LIN {X 0,Y 411.383,Z 368.831,A -85,B 0,C 180,E1 -10541.579,E2 -10541.579} C_VEL
LIN {X 0,Y 411.988,Z 360.367,A -85,B 0,C 180,E1 -10542.812,E2 -10542.812} C_VEL
LIN {X 0,Y 412.688,Z 350.209,A -85,B 0,C 180,E1 -10544.018,E2 -10544.018} C_VEL
LIN {X 0,Y 413.617,Z 338.309,A -85,B 0,C 180,E1 -10545.143,E2 -10545.143} C_VEL
LIN {X 0,Y 414.492,Z 326.832,A -85,B 0,C 180,E1 -10545.993,E2 -10545.993} C_VEL
LIN {X 0,Y 414.334,Z 319.686,A -85,B 0,C 180,E1 -10546.442,E2 -10546.442} C_VEL
LIN {X 0,Y 412.96,Z 306.533,A -85,B 0,C 180,E1 -10547.145,E2 -10547.145} C_VEL
LIN {X 0,Y 410.807,Z 293.982,A -85,B 0,C 180,E1 -10547.664,E2 -10547.664} C_VEL
LIN {X 0,Y 410.419,Z 291.596,A -85,B 0,C 180,E1 -10547.758,E2 -10547.758} C_VEL
LIN {X 0,Y 410.785,Z 283.542,A -85,B 0,C 180,E1 -10551.055,E2 -10551.055} C_VEL
LIN {X 0,Y 411.122,Z 276.006,A -85,B 0,C 180,E1 -10554.221,E2 -10554.221} C_VEL
LIN {X 0,Y 411.591,Z 268.703,A -85,B 0,C 180,E1 -10557.386,E2 -10557.386} C_VEL
LIN {X 0,Y 412.207,Z 261.207,A -85,B 0,C 180,E1 -10560.762,E2 -10560.762} C_VEL
LIN {X 0,Y 412.806,Z 255.521,A -85,B 0,C 180,E1 -10563.463,E2 -10563.463} C_VEL
LIN {X 0,Y 413.225,Z 250.596,A -85,B 0,C 180,E1 -10565.926,E2 -10565.926} C_VEL
LIN {X 0,Y 412.966,Z 247.13,A -85,B 0,C 180,E1 -10567.781,E2 -10567.781} C_VEL
LIN {X 0,Y 412.21,Z 242.601,A -85,B 0,C 180,E1 -10570.381,E2 -10570.381} C_VEL
LIN {X 0,Y 411.179,Z 237.269,A -85,B 0,C 180,E1 -10573.842,E2 -10573.842} C_VEL
LIN {X 0,Y 411.181,Z 237.269,A -85,B 0,C 180,E1 -10577.303,E2 -10577.303} C_VEL
LIN {X 0,Y 411.218,Z 237.265,A -85,B 0,C 180,E1 -10580.775,E2 -10580.775} C_VEL
LIN {X 0,Y 411.198,Z 237.268,A -85,B 0,C 180,E1 -10584.47,E2 -10584.47} C_VEL
LIN {X 0,Y 411.205,Z 237.267,A -85,B 0,C 180,E1 -10586.872,E2 -10586.872} C_VEL
LIN {X 0,Y 411.231,Z 237.262,A -85,B 0,C 180,E1 -10590.643,E2 -10590.643} C_VEL
LIN {X 0,Y 411.234,Z 237.263,A -85,B 0,C 180,E1 -10593.618,E2 -10593.618} C_VEL
LIN {X 0,Y 411.199,Z 237.267,A -85,B 0,C 180,E1 -10596.851,E2 -10596.851} C_VEL
LIN {X 0,Y 411.211,Z 237.264,A -85,B 0,C 180,E1 -10600.049,E2 -10600.049} C_VEL
LIN {X 0,Y 411.259,Z 237.257,A -85,B 0,C 180,E1 -10603.13,E2 -10603.13} C_VEL
LIN {X 0,Y 411.309,Z 237.253,A -85,B 0,C 180,E1 -10606.889,E2 -10606.889} C_VEL
LIN {X 0,Y 411.303,Z 237.253,A -85,B 0,C 180,E1 -10610.16,E2 -10610.16} C_VEL
LIN {X 0,Y 411.455,Z 237.234,A -85,B 0,C 180,E1 -10613.132,E2 -10613.132} C_VEL
LIN {X 0,Y 411.307,Z 237.254,A -85,B 0,C 180,E1 -10615.098,E2 -10615.098} C_VEL
LIN {X 0,Y 411.508,Z 237.228,A -85,B 0,C 180,E1 -10618.041,E2 -10618.041} C_VEL
LIN {X 0,Y 411.636,Z 237.212,A -85,B 0,C 180,E1 -10619.998,E2 -10619.998} C_VEL
LIN {X 0,Y 411.46,Z 237.235,A -85,B 0,C 180,E1 -10622.936,E2 -10622.936} C_VEL
LIN {X 0,Y 411.453,Z 237.233,A -85,B 0,C 180,E1 -10626.865,E2 -10626.865} C_VEL
LIN {X 0,Y 411.302,Z 237.254,A -85,B 0,C 180,E1 -10629.837,E2 -10629.837} C_VEL
LIN {X 0,Y 411.305,Z 237.254,A -85,B 0,C 180,E1 -10633.108,E2 -10633.108} C_VEL
LIN {X 0,Y 411.246,Z 237.264,A -85,B 0,C 180,E1 -10635.867,E2 -10635.867} C_VEL
LIN {X 0,Y 411,Z 237.293,A -85,B 0,C 180,E1 -10638.957,E2 -10638.957} C_VEL
LIN {X 0,Y 410.922,Z 237.508,A -85,B 0,C 180,E1 -10640.001,E2 -10640.001} C_VEL
LIN {X 0,Y 410.8,Z 240.356,A -85,B 0,C 180,E1 -10643.17,E2 -10643.17} C_VEL
LIN {X 0,Y 410.648,Z 243.385,A -85,B 0,C 180,E1 -10646.42,E2 -10646.42} C_VEL
LIN {X 0,Y 410.532,Z 246.522,A -85,B 0,C 180,E1 -10649.764,E2 -10649.764} C_VEL
LIN {X 0,Y 410.428,Z 249.88,A -85,B 0,C 180,E1 -10653.224,E2 -10653.224} C_VEL
LIN {X 0,Y 410.358,Z 251.98,A -85,B 0,C 180,E1 -10655.363,E2 -10655.363} C_VEL
LIN {X 0,Y 414.097,Z 265.764,A -85,B 0,C 180,E1 -10656.059,E2 -10656.059} C_VEL
LIN {X 0,Y 415.793,Z 273.443,A -85,B 0,C 180,E1 -10656.522,E2 -10656.522} C_VEL
LIN {X 0,Y 415.193,Z 285.886,A -85,B 0,C 180,E1 -10657.292,E2 -10657.292} C_VEL
LIN {X 0,Y 414.383,Z 297.741,A -85,B 0,C 180,E1 -10658.244,E2 -10658.244} C_VEL
LIN {X 0,Y 413.615,Z 309.082,A -85,B 0,C 180,E1 -10659.422,E2 -10659.422} C_VEL
LIN {X 0,Y 412.811,Z 319.31,A -85,B 0,C 180,E1 -10660.749,E2 -10660.749} C_VEL
LIN {X 0,Y 412.063,Z 327.701,A -85,B 0,C 180,E1 -10662.106,E2 -10662.106} C_VEL
LIN {X 0,Y 411.451,Z 335.153,A -85,B 0,C 180,E1 -10663.604,E2 -10663.604} C_VEL
LIN {X 0,Y 410.997,Z 340.674,A -85,B 0,C 180,E1 -10664.98,E2 -10664.98} C_VEL
LIN {X 0,Y 410.661,Z 345.143,A -85,B 0,C 180,E1 -10666.368,E2 -10666.368} C_VEL
LIN {X 0,Y 410.326,Z 349.345,A -85,B 0,C 180,E1 -10668.09,E2 -10668.09} C_VEL
LIN {X 0,Y 410.105,Z 351.57,A -85,B 0,C 180,E1 -10669.369,E2 -10669.369} C_VEL
LIN {X 0,Y 409.997,Z 353.106,A -85,B 0,C 180,E1 -10670.638,E2 -10670.638} C_VEL
LIN {X 0,Y 409.914,Z 353.998,A -85,B 0,C 180,E1 -10672.058,E2 -10672.058} C_VEL
LIN {X 0,Y 409.89,Z 354.02,A -85,B 0,C 180,E1 -10673.69,E2 -10673.69} C_VEL
LIN {X 0,Y 410.012,Z 352.684,A -85,B 0,C 180,E1 -10675.554,E2 -10675.554} C_VEL
LIN {X 0,Y 410.123,Z 350.484,A -85,B 0,C 180,E1 -10677.102,E2 -10677.102} C_VEL
LIN {X 0,Y 410.453,Z 346.63,A -85,B 0,C 180,E1 -10678.88,E2 -10678.88} C_VEL
LIN {X 0,Y 410.677,Z 342.631,A -85,B 0,C 180,E1 -10680.247,E2 -10680.247} C_VEL
LIN {X 0,Y 411.142,Z 336.186,A -85,B 0,C 180,E1 -10681.962,E2 -10681.962} C_VEL
LIN {X 0,Y 411.652,Z 329.265,A -85,B 0,C 180,E1 -10683.405,E2 -10683.405} C_VEL
LIN {X 0,Y 412.279,Z 321.13,A -85,B 0,C 180,E1 -10684.777,E2 -10684.777} C_VEL
LIN {X 0,Y 413.056,Z 311.428,A -85,B 0,C 180,E1 -10686.104,E2 -10686.104} C_VEL
LIN {X 0,Y 413.779,Z 300.81,A -85,B 0,C 180,E1 -10687.27,E2 -10687.27} C_VEL
LIN {X 0,Y 414.533,Z 289.167,A -85,B 0,C 180,E1 -10688.281,E2 -10688.281} C_VEL
LIN {X 0,Y 415.059,Z 277.707,A -85,B 0,C 180,E1 -10689.065,E2 -10689.065} C_VEL
LIN {X 0,Y 415.317,Z 273.033,A -85,B 0,C 180,E1 -10689.324,E2 -10689.324} C_VEL
LIN {X 0,Y 412.751,Z 260.609,A -85,B 0,C 180,E1 -10690.007,E2 -10690.007} C_VEL
LIN {X 0,Y 410.309,Z 250.786,A -85,B 0,C 180,E1 -10690.446,E2 -10690.446} C_VEL
LIN {X 0,Y 410.415,Z 246.968,A -85,B 0,C 180,E1 -10694.099,E2 -10694.099} C_VEL
LIN {X 0,Y 410.543,Z 242.824,A -85,B 0,C 180,E1 -10698.147,E2 -10698.147} C_VEL
LIN {X 0,Y 410.711,Z 238.835,A -85,B 0,C 180,E1 -10702.133,E2 -10702.133} C_VEL
LIN {X 0,Y 410.741,Z 237.852,A -85,B 0,C 180,E1 -10703.122,E2 -10703.122} C_VEL
LIN {X 0,Y 410.816,Z 237.314,A -85,B 0,C 180,E1 -10704.11,E2 -10704.11} C_VEL
LIN {X 0,Y 411.4,Z 237.239,A -85,B 0,C 180,E1 -10708.043,E2 -10708.043} C_VEL
LIN {X 0,Y 411.625,Z 237.211,A -85,B 0,C 180,E1 -10710.001,E2 -10710.001} C_VEL
LIN {X 0,Y 411.453,Z 237.233,A -85,B 0,C 180,E1 -10712.882,E2 -10712.882} C_VEL
LIN {X 0,Y 410.795,Z 237.321,A -85,B 0,C 180,E1 -10713.698,E2 -10713.698} C_VEL
LIN {X 0,Y 407.938,Z 237.68,A -85,B 0,C 180,E1 -10715.025,E2 -10715.025} C_VEL
LIN {X 0,Y 405.515,Z 237.979,A -85,B 0,C 180,E1 -10716.096,E2 -10716.096} C_VEL
LIN {X 0,Y 404.477,Z 238.104,A -85,B 0,C 180,E1 -10716.924,E2 -10716.924} C_VEL
LIN {X 0,Y 404.393,Z 238.112,A -85,B 0,C 180,E1 -10717.205,E2 -10717.205} C_VEL
LIN {X 0,Y 404.253,Z 238.132,A -85,B 0,C 180,E1 -10721.026,E2 -10721.026} C_VEL
LIN {X 0,Y 404.204,Z 238.134,A -85,B 0,C 180,E1 -10724.09,E2 -10724.09} C_VEL
LIN {X 0,Y 404.191,Z 238.139,A -85,B 0,C 180,E1 -10727.194,E2 -10727.194} C_VEL
LIN {X 0,Y 404.193,Z 238.137,A -85,B 0,C 180,E1 -10730.351,E2 -10730.351} C_VEL
LIN {X 0,Y 404.16,Z 238.14,A -85,B 0,C 180,E1 -10733.576,E2 -10733.576} C_VEL
LIN {X 0,Y 404.185,Z 238.141,A -85,B 0,C 180,E1 -10736.879,E2 -10736.879} C_VEL
LIN {X 0,Y 404.136,Z 238.144,A -85,B 0,C 180,E1 -10740.287,E2 -10740.287} C_VEL
LIN {X 0,Y 404.136,Z 238.143,A -85,B 0,C 180,E1 -10743.814,E2 -10743.814} C_VEL
LIN {X 0,Y 404.133,Z 238.147,A -85,B 0,C 180,E1 -10746.878,E2 -10746.878} C_VEL
LIN {X 0,Y 404.16,Z 238.141,A -85,B 0,C 180,E1 -10750.086,E2 -10750.086} C_VEL
LIN {X 0,Y 404.191,Z 238.137,A -85,B 0,C 180,E1 -10753.093,E2 -10753.093} C_VEL
LIN {X 0,Y 404.146,Z 238.142,A -85,B 0,C 180,E1 -10755.929,E2 -10755.929} C_VEL
LIN {X 0,Y 404.148,Z 238.145,A -85,B 0,C 180,E1 -10758.641,E2 -10758.641} C_VEL
LIN {X 0,Y 404.159,Z 238.139,A -85,B 0,C 180,E1 -10761.493,E2 -10761.493} C_VEL
LIN {X 0,Y 404.183,Z 238.138,A -85,B 0,C 180,E1 -10764.986,E2 -10764.986} C_VEL
LIN {X 0,Y 404.141,Z 238.146,A -85,B 0,C 180,E1 -10768.556,E2 -10768.556} C_VEL
LIN {X 0,Y 404.195,Z 238.138,A -85,B 0,C 180,E1 -10772.002,E2 -10772.002} C_VEL
LIN {X 0,Y 404.177,Z 238.137,A -85,B 0,C 180,E1 -10775.336,E2 -10775.336} C_VEL
LIN {X 0,Y 404.141,Z 238.145,A -85,B 0,C 180,E1 -10778.583,E2 -10778.583} C_VEL
LIN {X 0,Y 404.213,Z 238.136,A -85,B 0,C 180,E1 -10781.764,E2 -10781.764} C_VEL
LIN {X 0,Y 404.211,Z 238.134,A -85,B 0,C 180,E1 -10784.884,E2 -10784.884} C_VEL
LIN {X 0,Y 404.273,Z 238.129,A -85,B 0,C 180,E1 -10787.961,E2 -10787.961} C_VEL
LIN {X 0,Y 404.272,Z 238.126,A -85,B 0,C 180,E1 -10791,E2 -10791} C_VEL
LIN {X 0,Y 404.422,Z 238.111,A -85,B 0,C 180,E1 -10794.017,E2 -10794.017} C_VEL
LIN {X 0,Y 404.486,Z 238.102,A -85,B 0,C 180,E1 -10798.01,E2 -10798.01} C_VEL
LIN {X 0,Y 404.616,Z 238.086,A -85,B 0,C 180,E1 -10800.002,E2 -10800.002} C_VEL
LIN {X 0,Y 404.416,Z 238.108,A -85,B 0,C 180,E1 -10802.99,E2 -10802.99} C_VEL
LIN {X 0,Y 404.421,Z 238.11,A -85,B 0,C 180,E1 -10805.986,E2 -10805.986} C_VEL
LIN {X 0,Y 404.274,Z 238.126,A -85,B 0,C 180,E1 -10809.003,E2 -10809.003} C_VEL
LIN {X 0,Y 404.264,Z 238.129,A -85,B 0,C 180,E1 -10812.043,E2 -10812.043} C_VEL
LIN {X 0,Y 404.214,Z 238.136,A -85,B 0,C 180,E1 -10815.119,E2 -10815.119} C_VEL
LIN {X 0,Y 404.217,Z 238.133,A -85,B 0,C 180,E1 -10818.239,E2 -10818.239} C_VEL
LIN {X 0,Y 404.148,Z 238.145,A -85,B 0,C 180,E1 -10821.42,E2 -10821.42} C_VEL
LIN {X 0,Y 404.182,Z 238.138,A -85,B 0,C 180,E1 -10824.667,E2 -10824.667} C_VEL
LIN {X 0,Y 404.204,Z 238.135,A -85,B 0,C 180,E1 -10828,E2 -10828} C_VEL
LIN {X 0,Y 404.149,Z 238.144,A -85,B 0,C 180,E1 -10831.558,E2 -10831.558} C_VEL
LIN {X 0,Y 404.193,Z 238.139,A -85,B 0,C 180,E1 -10835.017,E2 -10835.017} C_VEL
LIN {X 0,Y 404.158,Z 238.143,A -85,B 0,C 180,E1 -10838.758,E2 -10838.758} C_VEL
LIN {X 0,Y 404.132,Z 238.145,A -85,B 0,C 180,E1 -10841.6,E2 -10841.6} C_VEL
LIN {X 0,Y 404.154,Z 238.142,A -85,B 0,C 180,E1 -10844.522,E2 -10844.522} C_VEL
LIN {X 0,Y 404.191,Z 238.256,A -85,B 0,C 180,E1 -10847.067,E2 -10847.067} C_VEL
LIN {X 0,Y 405.155,Z 243.672,A -85,B 0,C 180,E1 -10850.071,E2 -10850.071} C_VEL
LIN {X 0,Y 405.98,Z 248.823,A -85,B 0,C 180,E1 -10852.781,E2 -10852.781} C_VEL
LIN {X 0,Y 406.12,Z 252.109,A -85,B 0,C 180,E1 -10854.426,E2 -10854.426} C_VEL
LIN {X 0,Y 405.596,Z 258.634,A -85,B 0,C 180,E1 -10857.509,E2 -10857.509} C_VEL
LIN {X 0,Y 404.895,Z 266.103,A -85,B 0,C 180,E1 -10860.92,E2 -10860.92} C_VEL
LIN {X 0,Y 404.281,Z 274.615,A -85,B 0,C 180,E1 -10864.686,E2 -10864.686} C_VEL
LIN {X 0,Y 403.814,Z 282.385,A -85,B 0,C 180,E1 -10868.025,E2 -10868.025} C_VEL
LIN {X 0,Y 403.476,Z 289.938,A -85,B 0,C 180,E1 -10871.2,E2 -10871.2} C_VEL
LIN {X 0,Y 403.368,Z 292.457,A -85,B 0,C 180,E1 -10872.247,E2 -10872.247} C_VEL
LIN {X 0,Y 405.548,Z 306.349,A -85,B 0,C 180,E1 -10872.776,E2 -10872.776} C_VEL
LIN {X 0,Y 406.98,Z 318.757,A -85,B 0,C 180,E1 -10873.428,E2 -10873.428} C_VEL
LIN {X 0,Y 407.34,Z 325.761,A -85,B 0,C 180,E1 -10873.868,E2 -10873.868} C_VEL
LIN {X 0,Y 406.542,Z 337.384,A -85,B 0,C 180,E1 -10874.713,E2 -10874.713} C_VEL
LIN {X 0,Y 405.753,Z 348.11,A -85,B 0,C 180,E1 -10875.709,E2 -10875.709} C_VEL
LIN {X 0,Y 404.977,Z 358.889,A -85,B 0,C 180,E1 -10876.961,E2 -10876.961} C_VEL
LIN {X 0,Y 404.352,Z 367.659,A -85,B 0,C 180,E1 -10878.215,E2 -10878.215} C_VEL
LIN {X 0,Y 403.701,Z 376.182,A -85,B 0,C 180,E1 -10879.72,E2 -10879.72} C_VEL
LIN {X 0,Y 403.318,Z 383.032,A -85,B 0,C 180,E1 -10881.229,E2 -10881.229} C_VEL
LIN {X 0,Y 403.079,Z 389.323,A -85,B 0,C 180,E1 -10882.989,E2 -10882.989} C_VEL
LIN {X 0,Y 402.94,Z 393.407,A -85,B 0,C 180,E1 -10884.494,E2 -10884.494} C_VEL
LIN {X 0,Y 402.889,Z 396.421,A -85,B 0,C 180,E1 -10885.998,E2 -10885.998} C_VEL
LIN {X 0,Y 402.952,Z 397.892,A -85,B 0,C 180,E1 -10887,E2 -10887} C_VEL
LIN {X 0,Y 402.981,Z 398.918,A -85,B 0,C 180,E1 -10888,E2 -10888} C_VEL
LIN {X 0,Y 402.951,Z 399.544,A -85,B 0,C 180,E1 -10889,E2 -10889} C_VEL
LIN {X 0,Y 402.947,Z 399.779,A -85,B 0,C 180,E1 -10889.999,E2 -10889.999} C_VEL
LIN {X 0,Y 402.94,Z 399.595,A -85,B 0,C 180,E1 -10890.998,E2 -10890.998} C_VEL
LIN {X 0,Y 402.977,Z 398.986,A -85,B 0,C 180,E1 -10891.998,E2 -10891.998} C_VEL
LIN {X 0,Y 402.923,Z 397.978,A -85,B 0,C 180,E1 -10892.999,E2 -10892.999} C_VEL
LIN {X 0,Y 402.886,Z 396.569,A -85,B 0,C 180,E1 -10894,E2 -10894} C_VEL
LIN {X 0,Y 402.937,Z 393.613,A -85,B 0,C 180,E1 -10895.504,E2 -10895.504} C_VEL
LIN {X 0,Y 403.077,Z 389.618,A -85,B 0,C 180,E1 -10897.009,E2 -10897.009} C_VEL
LIN {X 0,Y 403.332,Z 383.501,A -85,B 0,C 180,E1 -10898.769,E2 -10898.769} C_VEL
LIN {X 0,Y 403.73,Z 376.805,A -85,B 0,C 180,E1 -10900.277,E2 -10900.277} C_VEL
LIN {X 0,Y 404.388,Z 368.518,A -85,B 0,C 180,E1 -10901.782,E2 -10901.782} C_VEL
LIN {X 0,Y 405.002,Z 360.071,A -85,B 0,C 180,E1 -10903.036,E2 -10903.036} C_VEL
LIN {X 0,Y 405.793,Z 349.715,A -85,B 0,C 180,E1 -10904.287,E2 -10904.287} C_VEL
LIN {X 0,Y 406.732,Z 338.09,A -85,B 0,C 180,E1 -10905.406,E2 -10905.406} C_VEL
LIN {X 0,Y 407.655,Z 326.793,A -85,B 0,C 180,E1 -10906.262,E2 -10906.262} C_VEL
LIN {X 0,Y 407.267,Z 317.779,A -85,B 0,C 180,E1 -10906.844,E2 -10906.844} C_VEL
LIN {X 0,Y 405.855,Z 304.954,A -85,B 0,C 180,E1 -10907.532,E2 -10907.532} C_VEL
LIN {X 0,Y 403.375,Z 291.178,A -85,B 0,C 180,E1 -10908.112,E2 -10908.112} C_VEL
LIN {X 0,Y 403.7,Z 284.484,A -85,B 0,C 180,E1 -10910.908,E2 -10910.908} C_VEL
LIN {X 0,Y 404.066,Z 276.963,A -85,B 0,C 180,E1 -10914.125,E2 -10914.125} C_VEL
LIN {X 0,Y 404.455,Z 270.807,A -85,B 0,C 180,E1 -10916.857,E2 -10916.857} C_VEL
LIN {X 0,Y 405.172,Z 262.271,A -85,B 0,C 180,E1 -10920.776,E2 -10920.776} C_VEL
LIN {X 0,Y 405.835,Z 256.06,A -85,B 0,C 180,E1 -10923.773,E2 -10923.773} C_VEL
LIN {X 0,Y 406.223,Z 251.626,A -85,B 0,C 180,E1 -10926.03,E2 -10926.03} C_VEL
LIN {X 0,Y 405.959,Z 248.21,A -85,B 0,C 180,E1 -10927.92,E2 -10927.92} C_VEL
LIN {X 0,Y 405.302,Z 244.18,A -85,B 0,C 180,E1 -10930.272,E2 -10930.272} C_VEL
LIN {X 0,Y 404.441,Z 239.708,A -85,B 0,C 180,E1 -10933.126,E2 -10933.126} C_VEL
LIN {X 0,Y 404.127,Z 238.148,A -85,B 0,C 180,E1 -10934.299,E2 -10934.299} C_VEL
LIN {X 0,Y 404.136,Z 238.147,A -85,B 0,C 180,E1 -10937.294,E2 -10937.294} C_VEL
LIN {X 0,Y 404.168,Z 238.143,A -85,B 0,C 180,E1 -10939.954,E2 -10939.954} C_VEL
LIN {X 0,Y 404.138,Z 238.147,A -85,B 0,C 180,E1 -10943.123,E2 -10943.123} C_VEL
LIN {X 0,Y 404.143,Z 238.145,A -85,B 0,C 180,E1 -10946.186,E2 -10946.186} C_VEL
LIN {X 0,Y 404.143,Z 238.145,A -85,B 0,C 180,E1 -10949.713,E2 -10949.713} C_VEL
LIN {X 0,Y 404.192,Z 238.139,A -85,B 0,C 180,E1 -10953.121,E2 -10953.121} C_VEL
LIN {X 0,Y 404.173,Z 238.141,A -85,B 0,C 180,E1 -10955.333,E2 -10955.333} C_VEL
LIN {X 0,Y 404.135,Z 238.145,A -85,B 0,C 180,E1 -10958.579,E2 -10958.579} C_VEL
LIN {X 0,Y 404.207,Z 238.137,A -85,B 0,C 180,E1 -10961.76,E2 -10961.76} C_VEL
LIN {X 0,Y 404.204,Z 238.138,A -85,B 0,C 180,E1 -10964.881,E2 -10964.881} C_VEL
LIN {X 0,Y 404.265,Z 238.13,A -85,B 0,C 180,E1 -10967.957,E2 -10967.957} C_VEL
LIN {X 0,Y 404.428,Z 238.109,A -85,B 0,C 180,E1 -10972.098,E2 -10972.098} C_VEL
LIN {X 0,Y 404.419,Z 238.111,A -85,B 0,C 180,E1 -10974.014,E2 -10974.014} C_VEL
LIN {X 0,Y 404.477,Z 238.103,A -85,B 0,C 180,E1 -10978.007,E2 -10978.007} C_VEL
LIN {X 0,Y 404.605,Z 238.087,A -85,B 0,C 180,E1 -10979.998,E2 -10979.998} C_VEL
LIN {X 0,Y 404.417,Z 238.112,A -85,B 0,C 180,E1 -10982.987,E2 -10982.987} C_VEL
LIN {X 0,Y 404.404,Z 238.11,A -85,B 0,C 180,E1 -10986.986,E2 -10986.986} C_VEL
LIN {X 0,Y 404.265,Z 238.13,A -85,B 0,C 180,E1 -10990.01,E2 -10990.01} C_VEL
LIN {X 0,Y 404.257,Z 238.133,A -85,B 0,C 180,E1 -10993.21,E2 -10993.21} C_VEL
LIN {X 0,Y 404.201,Z 238.142,A -85,B 0,C 180,E1 -10996.151,E2 -10996.151} C_VEL
LIN {X 0,Y 403.933,Z 238.173,A -85,B 0,C 180,E1 -10999.302,E2 -10999.302} C_VEL
LIN {X 0,Y 403.88,Z 238.8,A -85,B 0,C 180,E1 -11000.365,E2 -11000.365} C_VEL
LIN {X 0,Y 403.79,Z 240.868,A -85,B 0,C 180,E1 -11002.713,E2 -11002.713} C_VEL
LIN {X 0,Y 403.634,Z 243.684,A -85,B 0,C 180,E1 -11005.802,E2 -11005.802} C_VEL
LIN {X 0,Y 403.513,Z 247.059,A -85,B 0,C 180,E1 -11009.444,E2 -11009.444} C_VEL
LIN {X 0,Y 403.387,Z 250.162,A -85,B 0,C 180,E1 -11012.688,E2 -11012.688} C_VEL
LIN {X 0,Y 403.314,Z 252.404,A -85,B 0,C 180,E1 -11015.017,E2 -11015.017} C_VEL
LIN {X 0,Y 407.22,Z 266.7,A -85,B 0,C 180,E1 -11015.759,E2 -11015.759} C_VEL
LIN {X 0,Y 409.058,Z 274.822,A -85,B 0,C 180,E1 -11016.272,E2 -11016.272} C_VEL
LIN {X 0,Y 408.423,Z 286.701,A -85,B 0,C 180,E1 -11017.03,E2 -11017.03} C_VEL
LIN {X 0,Y 407.606,Z 297.859,A -85,B 0,C 180,E1 -11017.942,E2 -11017.942} C_VEL
LIN {X 0,Y 406.792,Z 309.043,A -85,B 0,C 180,E1 -11019.114,E2 -11019.114} C_VEL
LIN {X 0,Y 405.973,Z 318.81,A -85,B 0,C 180,E1 -11020.387,E2 -11020.387} C_VEL
LIN {X 0,Y 405.187,Z 327.424,A -85,B 0,C 180,E1 -11021.771,E2 -11021.771} C_VEL
LIN {X 0,Y 404.495,Z 335.464,A -85,B 0,C 180,E1 -11023.399,E2 -11023.399} C_VEL
LIN {X 0,Y 403.928,Z 341.95,A -85,B 0,C 180,E1 -11025.065,E2 -11025.065} C_VEL
LIN {X 0,Y 403.573,Z 346.249,A -85,B 0,C 180,E1 -11026.483,E2 -11026.483} C_VEL
LIN {X 0,Y 403.284,Z 349.498,A -85,B 0,C 180,E1 -11027.862,E2 -11027.862} C_VEL
LIN {X 0,Y 402.972,Z 352.698,A -85,B 0,C 180,E1 -11029.814,E2 -11029.814} C_VEL
LIN {X 0,Y 402.859,Z 354.265,A -85,B 0,C 180,E1 -11031.721,E2 -11031.721} C_VEL
LIN {X 0,Y 402.813,Z 354.431,A -85,B 0,C 180,E1 -11033.616,E2 -11033.616} C_VEL
LIN {X 0,Y 402.855,Z 353.571,A -85,B 0,C 180,E1 -11035.075,E2 -11035.075} C_VEL
LIN {X 0,Y 403.035,Z 351.436,A -85,B 0,C 180,E1 -11036.822,E2 -11036.822} C_VEL
LIN {X 0,Y 403.338,Z 347.863,A -85,B 0,C 180,E1 -11038.624,E2 -11038.624} C_VEL
LIN {X 0,Y 403.66,Z 342.49,A -85,B 0,C 180,E1 -11040.516,E2 -11040.516} C_VEL
LIN {X 0,Y 404.078,Z 336.992,A -85,B 0,C 180,E1 -11041.993,E2 -11041.993} C_VEL
LIN {X 0,Y 404.611,Z 330.337,A -85,B 0,C 180,E1 -11043.432,E2 -11043.432} C_VEL
LIN {X 0,Y 405.26,Z 322.165,A -85,B 0,C 180,E1 -11044.858,E2 -11044.858} C_VEL
LIN {X 0,Y 406.009,Z 313.063,A -85,B 0,C 180,E1 -11046.148,E2 -11046.148} C_VEL
LIN {X 0,Y 406.82,Z 302.177,A -85,B 0,C 180,E1 -11047.396,E2 -11047.396} C_VEL
LIN {X 0,Y 407.602,Z 290.65,A -85,B 0,C 180,E1 -11048.434,E2 -11048.434} C_VEL
LIN {X 0,Y 408.197,Z 278.538,A -85,B 0,C 180,E1 -11049.289,E2 -11049.289} C_VEL
LIN {X 0,Y 408.261,Z 272.641,A -85,B 0,C 180,E1 -11049.635,E2 -11049.635} C_VEL
LIN {X 0,Y 405.401,Z 259.949,A -85,B 0,C 180,E1 -11050.338,E2 -11050.338} C_VEL
LIN {X 0,Y 403.262,Z 251.152,A -85,B 0,C 180,E1 -11050.73,E2 -11050.73} C_VEL
LIN {X 0,Y 403.332,Z 247.963,A -85,B 0,C 180,E1 -11053.813,E2 -11053.813} C_VEL
LIN {X 0,Y 403.443,Z 244.439,A -85,B 0,C 180,E1 -11057.286,E2 -11057.286} C_VEL
LIN {X 0,Y 403.551,Z 240.737,A -85,B 0,C 180,E1 -11060.983,E2 -11060.983} C_VEL
LIN {X 0,Y 403.716,Z 238.739,A -85,B 0,C 180,E1 -11063.002,E2 -11063.002} C_VEL
LIN {X 0,Y 403.749,Z 238.194,A -85,B 0,C 180,E1 -11064.006,E2 -11064.006} C_VEL
LIN {X 0,Y 403.871,Z 238.178,A -85,B 0,C 180,E1 -11066.01,E2 -11066.01} C_VEL
LIN {X 0,Y 404.359,Z 238.116,A -85,B 0,C 180,E1 -11068.009,E2 -11068.009} C_VEL
LIN {X 0,Y 404.595,Z 238.087,A -85,B 0,C 180,E1 -11070.001,E2 -11070.001} C_VEL
LIN {X 0,Y 404.411,Z 238.111,A -85,B 0,C 180,E1 -11072.989,E2 -11072.989} C_VEL
LIN {X 0,Y 404.398,Z 238.113,A -85,B 0,C 180,E1 -11076.988,E2 -11076.988} C_VEL
LIN {X 0,Y 404.393,Z 238.112,A -85,B 0,C 180,E1 -11077.205,E2 -11077.205} C_VEL
LIN {X 0,Y 403.714,Z 238.196,A -85,B 0,C 180,E1 -11078.035,E2 -11078.035} C_VEL
LIN {X 0,Y 400.797,Z 238.563,A -85,B 0,C 180,E1 -11079.384,E2 -11079.384} C_VEL
LIN {X 0,Y 398.329,Z 238.871,A -85,B 0,C 180,E1 -11080.473,E2 -11080.473} C_VEL
LIN {X 0,Y 397.275,Z 239.001,A -85,B 0,C 180,E1 -11081.317,E2 -11081.317} C_VEL
LIN {X 0,Y 397.192,Z 239.008,A -85,B 0,C 180,E1 -11081.603,E2 -11081.603} C_VEL
LIN {X 0,Y 397.168,Z 239.011,A -85,B 0,C 180,E1 -11084.344,E2 -11084.344} C_VEL
LIN {X 0,Y 397.163,Z 239.013,A -85,B 0,C 180,E1 -11087.508,E2 -11087.508} C_VEL
LIN {X 0,Y 397.142,Z 239.017,A -85,B 0,C 180,E1 -11090.729,E2 -11090.729} C_VEL
LIN {X 0,Y 397.123,Z 239.016,A -85,B 0,C 180,E1 -11094.02,E2 -11094.02} C_VEL
LIN {X 0,Y 397.184,Z 239.01,A -85,B 0,C 180,E1 -11097.392,E2 -11097.392} C_VEL
LIN {X 0,Y 397.069,Z 239.027,A -85,B 0,C 180,E1 -11100.884,E2 -11100.884} C_VEL
LIN {X 0,Y 397.117,Z 239.02,A -85,B 0,C 180,E1 -11104.495,E2 -11104.495} C_VEL
LIN {X 0,Y 397.102,Z 239.021,A -85,B 0,C 180,E1 -11108.276,E2 -11108.276} C_VEL
LIN {X 0,Y 397.149,Z 239.014,A -85,B 0,C 180,E1 -11111.995,E2 -11111.995} C_VEL
LIN {X 0,Y 397.105,Z 239.02,A -85,B 0,C 180,E1 -11115.068,E2 -11115.068} C_VEL
LIN {X 0,Y 397.105,Z 239.02,A -85,B 0,C 180,E1 -11118.016,E2 -11118.016} C_VEL
LIN {X 0,Y 397.134,Z 239.015,A -85,B 0,C 180,E1 -11121.139,E2 -11121.139} C_VEL
LIN {X 0,Y 397.118,Z 239.021,A -85,B 0,C 180,E1 -11124.499,E2 -11124.499} C_VEL
LIN {X 0,Y 397.077,Z 239.024,A -85,B 0,C 180,E1 -11127.931,E2 -11127.931} C_VEL
LIN {X 0,Y 397.121,Z 239.017,A -85,B 0,C 180,E1 -11131.459,E2 -11131.459} C_VEL
LIN {X 0,Y 397.153,Z 239.016,A -85,B 0,C 180,E1 -11134.49,E2 -11134.49} C_VEL
LIN {X 0,Y 397.11,Z 239.018,A -85,B 0,C 180,E1 -11137.088,E2 -11137.088} C_VEL
LIN {X 0,Y 397.15,Z 239.016,A -85,B 0,C 180,E1 -11140.355,E2 -11140.355} C_VEL
LIN {X 0,Y 397.17,Z 239.012,A -85,B 0,C 180,E1 -11143.555,E2 -11143.555} C_VEL
LIN {X 0,Y 397.233,Z 239.003,A -85,B 0,C 180,E1 -11146.705,E2 -11146.705} C_VEL
LIN {X 0,Y 397.226,Z 239.008,A -85,B 0,C 180,E1 -11149.811,E2 -11149.811} C_VEL
LIN {X 0,Y 397.34,Z 238.989,A -85,B 0,C 180,E1 -11152.889,E2 -11152.889} C_VEL
LIN {X 0,Y 397.257,Z 238.999,A -85,B 0,C 180,E1 -11154.927,E2 -11154.927} C_VEL
LIN {X 0,Y 397.455,Z 238.978,A -85,B 0,C 180,E1 -11157.975,E2 -11157.975} C_VEL
LIN {X 0,Y 397.586,Z 238.962,A -85,B 0,C 180,E1 -11160.002,E2 -11160.002} C_VEL
LIN {X 0,Y 397.375,Z 238.985,A -85,B 0,C 180,E1 -11163.043,E2 -11163.043} C_VEL
LIN {X 0,Y 397.371,Z 238.988,A -85,B 0,C 180,E1 -11166.093,E2 -11166.093} C_VEL
LIN {X 0,Y 397.244,Z 239.003,A -85,B 0,C 180,E1 -11169.164,E2 -11169.164} C_VEL
LIN {X 0,Y 397.228,Z 239.004,A -85,B 0,C 180,E1 -11172.259,E2 -11172.259} C_VEL
LIN {X 0,Y 397.187,Z 239.012,A -85,B 0,C 180,E1 -11175.393,E2 -11175.393} C_VEL
LIN {X 0,Y 397.17,Z 239.01,A -85,B 0,C 180,E1 -11178.574,E2 -11178.574} C_VEL
LIN {X 0,Y 397.106,Z 239.02,A -85,B 0,C 180,E1 -11181.819,E2 -11181.819} C_VEL
LIN {X 0,Y 397.164,Z 239.015,A -85,B 0,C 180,E1 -11185.132,E2 -11185.132} C_VEL
LIN {X 0,Y 397.171,Z 239.012,A -85,B 0,C 180,E1 -11187.776,E2 -11187.776} C_VEL
LIN {X 0,Y 397.088,Z 239.023,A -85,B 0,C 180,E1 -11190.883,E2 -11190.883} C_VEL
LIN {X 0,Y 397.134,Z 239.016,A -85,B 0,C 180,E1 -11194.494,E2 -11194.494} C_VEL
LIN {X 0,Y 397.108,Z 239.018,A -85,B 0,C 180,E1 -11198.276,E2 -11198.276} C_VEL
LIN {X 0,Y 397.098,Z 239.023,A -85,B 0,C 180,E1 -11200.909,E2 -11200.909} C_VEL
LIN {X 0,Y 397.11,Z 239.02,A -85,B 0,C 180,E1 -11203.649,E2 -11203.649} C_VEL
LIN {X 0,Y 397.19,Z 239.219,A -85,B 0,C 180,E1 -11206.82,E2 -11206.82} C_VEL
LIN {X 0,Y 398.159,Z 244.835,A -85,B 0,C 180,E1 -11209.991,E2 -11209.991} C_VEL
LIN {X 0,Y 398.916,Z 249.382,A -85,B 0,C 180,E1 -11212.449,E2 -11212.449} C_VEL
LIN {X 0,Y 399.091,Z 253.353,A -85,B 0,C 180,E1 -11214.469,E2 -11214.469} C_VEL
LIN {X 0,Y 398.577,Z 259.448,A -85,B 0,C 180,E1 -11217.415,E2 -11217.415} C_VEL
LIN {X 0,Y 397.833,Z 267.023,A -85,B 0,C 180,E1 -11220.934,E2 -11220.934} C_VEL
LIN {X 0,Y 397.238,Z 274.839,A -85,B 0,C 180,E1 -11224.464,E2 -11224.464} C_VEL
LIN {X 0,Y 396.806,Z 282.02,A -85,B 0,C 180,E1 -11227.616,E2 -11227.616} C_VEL
LIN {X 0,Y 396.423,Z 289.504,A -85,B 0,C 180,E1 -11230.853,E2 -11230.853} C_VEL
LIN {X 0,Y 396.305,Z 292.251,A -85,B 0,C 180,E1 -11231.954,E2 -11231.954} C_VEL
LIN {X 0,Y 398.487,Z 305.801,A -85,B 0,C 180,E1 -11232.479,E2 -11232.479} C_VEL
LIN {X 0,Y 399.995,Z 318.739,A -85,B 0,C 180,E1 -11233.176,E2 -11233.176} C_VEL
LIN {X 0,Y 400.404,Z 326.638,A -85,B 0,C 180,E1 -11233.689,E2 -11233.689} C_VEL
LIN {X 0,Y 399.548,Z 338.18,A -85,B 0,C 180,E1 -11234.57,E2 -11234.57} C_VEL
LIN {X 0,Y 398.632,Z 349.854,A -85,B 0,C 180,E1 -11235.709,E2 -11235.709} C_VEL
LIN {X 0,Y 398.039,Z 358.317,A -85,B 0,C 180,E1 -11236.729,E2 -11236.729} C_VEL
LIN {X 0,Y 397.365,Z 367.116,A -85,B 0,C 180,E1 -11238.005,E2 -11238.005} C_VEL
LIN {X 0,Y 396.653,Z 375.674,A -85,B 0,C 180,E1 -11239.535,E2 -11239.535} C_VEL
LIN {X 0,Y 396.238,Z 382.544,A -85,B 0,C 180,E1 -11241.071,E2 -11241.071} C_VEL
LIN {X 0,Y 396.007,Z 388.856,A -85,B 0,C 180,E1 -11242.863,E2 -11242.863} C_VEL
LIN {X 0,Y 395.842,Z 392.431,A -85,B 0,C 180,E1 -11244.181,E2 -11244.181} C_VEL
LIN {X 0,Y 395.811,Z 395.986,A -85,B 0,C 180,E1 -11245.926,E2 -11245.926} C_VEL
LIN {X 0,Y 395.852,Z 397.47,A -85,B 0,C 180,E1 -11246.946,E2 -11246.946} C_VEL
LIN {X 0,Y 395.91,Z 398.504,A -85,B 0,C 180,E1 -11247.964,E2 -11247.964} C_VEL
LIN {X 0,Y 395.876,Z 399.136,A -85,B 0,C 180,E1 -11248.982,E2 -11248.982} C_VEL
LIN {X 0,Y 395.869,Z 399.376,A -85,B 0,C 180,E1 -11249.999,E2 -11249.999} C_VEL
LIN {X 0,Y 395.865,Z 399.204,A -85,B 0,C 180,E1 -11251.016,E2 -11251.016} C_VEL
LIN {X 0,Y 395.906,Z 398.601,A -85,B 0,C 180,E1 -11252.034,E2 -11252.034} C_VEL
LIN {X 0,Y 395.807,Z 396.192,A -85,B 0,C 180,E1 -11254.072,E2 -11254.072} C_VEL
LIN {X 0,Y 395.838,Z 392.774,A -85,B 0,C 180,E1 -11255.815,E2 -11255.815} C_VEL
LIN {X 0,Y 396.057,Z 387.675,A -85,B 0,C 180,E1 -11257.647,E2 -11257.647} C_VEL
LIN {X 0,Y 396.394,Z 381.101,A -85,B 0,C 180,E1 -11259.438,E2 -11259.438} C_VEL
LIN {X 0,Y 396.87,Z 373.933,A -85,B 0,C 180,E1 -11260.973,E2 -11260.973} C_VEL
LIN {X 0,Y 397.721,Z 365.029,A -85,B 0,C 180,E1 -11262.5,E2 -11262.5} C_VEL
LIN {X 0,Y 398.472,Z 355.104,A -85,B 0,C 180,E1 -11263.884,E2 -11263.884} C_VEL
LIN {X 0,Y 399.307,Z 344.704,A -85,B 0,C 180,E1 -11265.046,E2 -11265.046} C_VEL
LIN {X 0,Y 400.286,Z 333.412,A -85,B 0,C 180,E1 -11266.052,E2 -11266.052} C_VEL
LIN {X 0,Y 400.854,Z 325.047,A -85,B 0,C 180,E1 -11266.662,E2 -11266.662} C_VEL
LIN {X 0,Y 399.796,Z 312.078,A -85,B 0,C 180,E1 -11267.483,E2 -11267.483} C_VEL
LIN {X 0,Y 398.039,Z 299.942,A -85,B 0,C 180,E1 -11268.092,E2 -11268.092} C_VEL
LIN {X 0,Y 396.333,Z 290.751,A -85,B 0,C 180,E1 -11268.478,E2 -11268.478} C_VEL
LIN {X 0,Y 396.716,Z 282.917,A -85,B 0,C 180,E1 -11271.839,E2 -11271.839} C_VEL
LIN {X 0,Y 397.221,Z 274.584,A -85,B 0,C 180,E1 -11275.531,E2 -11275.531} C_VEL
LIN {X 0,Y 397.765,Z 266.879,A -85,B 0,C 180,E1 -11279.07,E2 -11279.07} C_VEL
LIN {X 0,Y 398.456,Z 260.456,A -85,B 0,C 180,E1 -11282.152,E2 -11282.152} C_VEL
LIN {X 0,Y 399.073,Z 255.006,A -85,B 0,C 180,E1 -11284.913,E2 -11284.913} C_VEL
LIN {X 0,Y 399.204,Z 251.552,A -85,B 0,C 180,E1 -11286.766,E2 -11286.766} C_VEL
LIN {X 0,Y 398.561,Z 247.021,A -85,B 0,C 180,E1 -11289.404,E2 -11289.404} C_VEL
LIN {X 0,Y 397.739,Z 242.598,A -85,B 0,C 180,E1 -11292.178,E2 -11292.178} C_VEL
LIN {X 0,Y 397.097,Z 239.024,A -85,B 0,C 180,E1 -11294.763,E2 -11294.763} C_VEL
LIN {X 0,Y 397.065,Z 239.028,A -85,B 0,C 180,E1 -11298.02,E2 -11298.02} C_VEL
LIN {X 0,Y 397.13,Z 239.02,A -85,B 0,C 180,E1 -11301.137,E2 -11301.137} C_VEL
LIN {X 0,Y 397.119,Z 239.022,A -85,B 0,C 180,E1 -11304.495,E2 -11304.495} C_VEL
LIN {X 0,Y 397.077,Z 239.027,A -85,B 0,C 180,E1 -11307.927,E2 -11307.927} C_VEL
LIN {X 0,Y 397.12,Z 239.021,A -85,B 0,C 180,E1 -11311.455,E2 -11311.455} C_VEL
LIN {X 0,Y 397.149,Z 239.017,A -85,B 0,C 180,E1 -11314.486,E2 -11314.486} C_VEL
LIN {X 0,Y 397.105,Z 239.022,A -85,B 0,C 180,E1 -11317.084,E2 -11317.084} C_VEL
LIN {X 0,Y 397.145,Z 239.017,A -85,B 0,C 180,E1 -11320.351,E2 -11320.351} C_VEL
LIN {X 0,Y 397.162,Z 239.014,A -85,B 0,C 180,E1 -11323.552,E2 -11323.552} C_VEL
LIN {X 0,Y 397.224,Z 239.007,A -85,B 0,C 180,E1 -11326.701,E2 -11326.701} C_VEL
LIN {X 0,Y 397.224,Z 239.006,A -85,B 0,C 180,E1 -11329.808,E2 -11329.808} C_VEL
LIN {X 0,Y 397.359,Z 238.99,A -85,B 0,C 180,E1 -11332.887,E2 -11332.887} C_VEL
LIN {X 0,Y 397.251,Z 239.004,A -85,B 0,C 180,E1 -11334.924,E2 -11334.924} C_VEL
LIN {X 0,Y 397.446,Z 238.979,A -85,B 0,C 180,E1 -11337.972,E2 -11337.972} C_VEL
LIN {X 0,Y 397.574,Z 238.963,A -85,B 0,C 180,E1 -11339.998,E2 -11339.998} C_VEL
LIN {X 0,Y 397.376,Z 238.989,A -85,B 0,C 180,E1 -11343.04,E2 -11343.04} C_VEL
LIN {X 0,Y 397.356,Z 238.988,A -85,B 0,C 180,E1 -11347.11,E2 -11347.11} C_VEL
LIN {X 0,Y 397.223,Z 239.006,A -85,B 0,C 180,E1 -11350.189,E2 -11350.189} C_VEL
LIN {X 0,Y 397.217,Z 239.01,A -85,B 0,C 180,E1 -11353.32,E2 -11353.32} C_VEL
LIN {X 0,Y 397.128,Z 239.024,A -85,B 0,C 180,E1 -11356.447,E2 -11356.447} C_VEL
LIN {X 0,Y 396.86,Z 239.151,A -85,B 0,C 180,E1 -11359.66,E2 -11359.66} C_VEL
LIN {X 0,Y 396.734,Z 242.008,A -85,B 0,C 180,E1 -11362.935,E2 -11362.935} C_VEL
LIN {X 0,Y 396.567,Z 245.036,A -85,B 0,C 180,E1 -11366.297,E2 -11366.297} C_VEL
LIN {X 0,Y 396.44,Z 248.215,A -85,B 0,C 180,E1 -11369.758,E2 -11369.758} C_VEL
LIN {X 0,Y 396.308,Z 251.591,A -85,B 0,C 180,E1 -11373.347,E2 -11373.347} C_VEL
LIN {X 0,Y 396.264,Z 252.842,A -85,B 0,C 180,E1 -11374.65,E2 -11374.65} C_VEL
LIN {X 0,Y 400.425,Z 267.794,A -85,B 0,C 180,E1 -11375.46,E2 -11375.46} C_VEL
LIN {X 0,Y 402.286,Z 276.884,A -85,B 0,C 180,E1 -11376.054,E2 -11376.054} C_VEL
LIN {X 0,Y 401.573,Z 288.465,A -85,B 0,C 180,E1 -11376.826,E2 -11376.826} C_VEL
LIN {X 0,Y 400.717,Z 299.527,A -85,B 0,C 180,E1 -11377.775,E2 -11377.775} C_VEL
LIN {X 0,Y 399.895,Z 310.096,A -85,B 0,C 180,E1 -11378.922,E2 -11378.922} C_VEL
LIN {X 0,Y 399.071,Z 319.607,A -85,B 0,C 180,E1 -11380.196,E2 -11380.196} C_VEL
LIN {X 0,Y 398.335,Z 327.141,A -85,B 0,C 180,E1 -11381.425,E2 -11381.425} C_VEL
LIN {X 0,Y 397.665,Z 334.277,A -85,B 0,C 180,E1 -11382.837,E2 -11382.837} C_VEL
LIN {X 0,Y 397.133,Z 340.112,A -85,B 0,C 180,E1 -11384.26,E2 -11384.26} C_VEL
LIN {X 0,Y 396.656,Z 344.823,A -85,B 0,C 180,E1 -11385.683,E2 -11385.683} C_VEL
LIN {X 0,Y 396.374,Z 348.564,A -85,B 0,C 180,E1 -11387.122,E2 -11387.122} C_VEL
LIN {X 0,Y 396.021,Z 352.048,A -85,B 0,C 180,E1 -11388.959,E2 -11388.959} C_VEL
LIN {X 0,Y 395.845,Z 353.673,A -85,B 0,C 180,E1 -11390.272,E2 -11390.272} C_VEL
LIN {X 0,Y 395.788,Z 354.623,A -85,B 0,C 180,E1 -11391.576,E2 -11391.576} C_VEL
LIN {X 0,Y 395.707,Z 354.936,A -85,B 0,C 180,E1 -11393.053,E2 -11393.053} C_VEL
LIN {X 0,Y 395.755,Z 354.228,A -85,B 0,C 180,E1 -11394.771,E2 -11394.771} C_VEL
LIN {X 0,Y 395.934,Z 352.196,A -85,B 0,C 180,E1 -11396.616,E2 -11396.616} C_VEL
LIN {X 0,Y 396.201,Z 349.016,A -85,B 0,C 180,E1 -11398.365,E2 -11398.365} C_VEL
LIN {X 0,Y 396.553,Z 344.013,A -85,B 0,C 180,E1 -11400.27,E2 -11400.27} C_VEL
LIN {X 0,Y 396.991,Z 338.368,A -85,B 0,C 180,E1 -11401.88,E2 -11401.88} C_VEL
LIN {X 0,Y 397.582,Z 331.218,A -85,B 0,C 180,E1 -11403.492,E2 -11403.492} C_VEL
LIN {X 0,Y 398.244,Z 323.199,A -85,B 0,C 180,E1 -11404.943,E2 -11404.943} C_VEL
LIN {X 0,Y 399.061,Z 313.778,A -85,B 0,C 180,E1 -11406.312,E2 -11406.312} C_VEL
LIN {X 0,Y 399.853,Z 303.487,A -85,B 0,C 180,E1 -11407.526,E2 -11407.526} C_VEL
LIN {X 0,Y 400.602,Z 292.89,A -85,B 0,C 180,E1 -11408.531,E2 -11408.531} C_VEL
LIN {X 0,Y 401.268,Z 280.801,A -85,B 0,C 180,E1 -11409.429,E2 -11409.429} C_VEL
LIN {X 0,Y 401.566,Z 275.177,A -85,B 0,C 180,E1 -11409.77,E2 -11409.77} C_VEL
LIN {X 0,Y 398.952,Z 262.645,A -85,B 0,C 180,E1 -11410.513,E2 -11410.513} C_VEL
LIN {X 0,Y 396.18,Z 251.501,A -85,B 0,C 180,E1 -11411.044,E2 -11411.044} C_VEL
LIN {X 0,Y 396.246,Z 247.908,A -85,B 0,C 180,E1 -11414.572,E2 -11414.572} C_VEL
LIN {X 0,Y 396.385,Z 244.728,A -85,B 0,C 180,E1 -11417.717,E2 -11417.717} C_VEL
LIN {X 0,Y 396.575,Z 240.645,A -85,B 0,C 180,E1 -11421.851,E2 -11421.851} C_VEL
LIN {X 0,Y 396.653,Z 239.642,A -85,B 0,C 180,E1 -11422.876,E2 -11422.876} C_VEL
LIN {X 0,Y 396.687,Z 239.074,A -85,B 0,C 180,E1 -11423.899,E2 -11423.899} C_VEL
LIN {X 0,Y 396.827,Z 239.056,A -85,B 0,C 180,E1 -11425.939,E2 -11425.939} C_VEL
LIN {X 0,Y 397.293,Z 238.996,A -85,B 0,C 180,E1 -11427.974,E2 -11427.974} C_VEL
LIN {X 0,Y 397.564,Z 238.962,A -85,B 0,C 180,E1 -11430.001,E2 -11430.001} C_VEL
LIN {X 0,Y 397.369,Z 238.989,A -85,B 0,C 180,E1 -11433.042,E2 -11433.042} C_VEL
LIN {X 0,Y 397.35,Z 238.992,A -85,B 0,C 180,E1 -11437.113,E2 -11437.113} C_VEL
LIN {X 0,Y 397.217,Z 239.004,A -85,B 0,C 180,E1 -11440.192,E2 -11440.192} C_VEL
LIN {X 0,Y 397.192,Z 239.008,A -85,B 0,C 180,E1 -11441.603,E2 -11441.603} C_VEL
LIN {X 0,Y 396.53,Z 239.092,A -85,B 0,C 180,E1 -11442.449,E2 -11442.449} C_VEL
LIN {X 0,Y 393.669,Z 239.447,A -85,B 0,C 180,E1 -11443.825,E2 -11443.825} C_VEL
LIN {X 0,Y 391.242,Z 239.753,A -85,B 0,C 180,E1 -11444.936,E2 -11444.936} C_VEL
LIN {X 0,Y 390.197,Z 239.879,A -85,B 0,C 180,E1 -11445.796,E2 -11445.796} C_VEL
LIN {X 0,Y 390.111,Z 239.889,A -85,B 0,C 180,E1 -11446.087,E2 -11446.087} C_VEL
LIN {X 0,Y 390.108,Z 239.894,A -85,B 0,C 180,E1 -11448.923,E2 -11448.923} C_VEL
LIN {X 0,Y 390.054,Z 239.897,A -85,B 0,C 180,E1 -11452.234,E2 -11452.234} C_VEL
LIN {X 0,Y 390.109,Z 239.89,A -85,B 0,C 180,E1 -11455.745,E2 -11455.745} C_VEL
LIN {X 0,Y 390.049,Z 239.9,A -85,B 0,C 180,E1 -11459.111,E2 -11459.111} C_VEL
LIN {X 0,Y 390.034,Z 239.904,A -85,B 0,C 180,E1 -11462.723,E2 -11462.723} C_VEL
LIN {X 0,Y 390.049,Z 239.897,A -85,B 0,C 180,E1 -11465.828,E2 -11465.828} C_VEL
LIN {X 0,Y 390.067,Z 239.896,A -85,B 0,C 180,E1 -11469.221,E2 -11469.221} C_VEL
LIN {X 0,Y 390.114,Z 239.893,A -85,B 0,C 180,E1 -11472.389,E2 -11472.389} C_VEL
LIN {X 0,Y 390.056,Z 239.896,A -85,B 0,C 180,E1 -11475.359,E2 -11475.359} C_VEL
LIN {X 0,Y 390.064,Z 239.899,A -85,B 0,C 180,E1 -11478.194,E2 -11478.194} C_VEL
LIN {X 0,Y 390.092,Z 239.894,A -85,B 0,C 180,E1 -11480.911,E2 -11480.911} C_VEL
LIN {X 0,Y 390.083,Z 239.895,A -85,B 0,C 180,E1 -11484.795,E2 -11484.795} C_VEL
LIN {X 0,Y 390.022,Z 239.905,A -85,B 0,C 180,E1 -11488.498,E2 -11488.498} C_VEL
LIN {X 0,Y 390.117,Z 239.892,A -85,B 0,C 180,E1 -11492.072,E2 -11492.072} C_VEL
LIN {X 0,Y 390.08,Z 239.894,A -85,B 0,C 180,E1 -11495.521,E2 -11495.521} C_VEL
LIN {X 0,Y 390.058,Z 239.897,A -85,B 0,C 180,E1 -11498.88,E2 -11498.88} C_VEL
LIN {X 0,Y 390.131,Z 239.891,A -85,B 0,C 180,E1 -11502.169,E2 -11502.169} C_VEL
LIN {X 0,Y 390.151,Z 239.886,A -85,B 0,C 180,E1 -11505.395,E2 -11505.395} C_VEL
LIN {X 0,Y 390.162,Z 239.884,A -85,B 0,C 180,E1 -11508.573,E2 -11508.573} C_VEL
LIN {X 0,Y 390.275,Z 239.873,A -85,B 0,C 180,E1 -11512.073,E2 -11512.073} C_VEL
LIN {X 0,Y 390.229,Z 239.874,A -85,B 0,C 180,E1 -11514.835,E2 -11514.835} C_VEL
LIN {X 0,Y 390.424,Z 239.854,A -85,B 0,C 180,E1 -11517.938,E2 -11517.938} C_VEL
LIN {X 0,Y 390.555,Z 239.837,A -85,B 0,C 180,E1 -11520.002,E2 -11520.002} C_VEL
LIN {X 0,Y 390.31,Z 239.865,A -85,B 0,C 180,E1 -11523.098,E2 -11523.098} C_VEL
LIN {X 0,Y 390.324,Z 239.864,A -85,B 0,C 180,E1 -11526.203,E2 -11526.203} C_VEL
LIN {X 0,Y 390.201,Z 239.882,A -85,B 0,C 180,E1 -11529.33,E2 -11529.33} C_VEL
LIN {X 0,Y 390.179,Z 239.881,A -85,B 0,C 180,E1 -11532.484,E2 -11532.484} C_VEL
LIN {X 0,Y 390.148,Z 239.889,A -85,B 0,C 180,E1 -11535.678,E2 -11535.678} C_VEL
LIN {X 0,Y 390.114,Z 239.891,A -85,B 0,C 180,E1 -11538.923,E2 -11538.923} C_VEL
LIN {X 0,Y 390.049,Z 239.897,A -85,B 0,C 180,E1 -11542.235,E2 -11542.235} C_VEL
LIN {X 0,Y 390.127,Z 239.89,A -85,B 0,C 180,E1 -11545.743,E2 -11545.743} C_VEL
LIN {X 0,Y 390.068,Z 239.899,A -85,B 0,C 180,E1 -11549.11,E2 -11549.11} C_VEL
LIN {X 0,Y 390.052,Z 239.899,A -85,B 0,C 180,E1 -11552.722,E2 -11552.722} C_VEL
LIN {X 0,Y 390.065,Z 239.896,A -85,B 0,C 180,E1 -11555.825,E2 -11555.825} C_VEL
LIN {X 0,Y 390.076,Z 239.898,A -85,B 0,C 180,E1 -11559.218,E2 -11559.218} C_VEL
LIN {X 0,Y 390.052,Z 239.901,A -85,B 0,C 180,E1 -11562.374,E2 -11562.374} C_VEL
LIN {X 0,Y 390.055,Z 239.897,A -85,B 0,C 180,E1 -11565.355,E2 -11565.355} C_VEL
LIN {X 0,Y 390.107,Z 240.013,A -85,B 0,C 180,E1 -11566.47,E2 -11566.47} C_VEL
LIN {X 0,Y 391.086,Z 245.565,A -85,B 0,C 180,E1 -11569.688,E2 -11569.688} C_VEL
LIN {X 0,Y 392.084,Z 251.795,A -85,B 0,C 180,E1 -11573.095,E2 -11573.095} C_VEL
LIN {X 0,Y 391.94,Z 256.708,A -85,B 0,C 180,E1 -11575.574,E2 -11575.574} C_VEL
LIN {X 0,Y 391.14,Z 264.13,A -85,B 0,C 180,E1 -11579.167,E2 -11579.167} C_VEL
LIN {X 0,Y 390.483,Z 271.652,A -85,B 0,C 180,E1 -11582.679,E2 -11582.679} C_VEL
LIN {X 0,Y 389.961,Z 279.118,A -85,B 0,C 180,E1 -11586.076,E2 -11586.076} C_VEL
LIN {X 0,Y 389.47,Z 287.851,A -85,B 0,C 180,E1 -11589.948,E2 -11589.948} C_VEL
LIN {X 0,Y 389.251,Z 291.892,A -85,B 0,C 180,E1 -11591.648,E2 -11591.648} C_VEL
LIN {X 0,Y 391.428,Z 305.184,A -85,B 0,C 180,E1 -11592.172,E2 -11592.172} C_VEL
LIN {X 0,Y 393.008,Z 318.66,A -85,B 0,C 180,E1 -11592.912,E2 -11592.912} C_VEL
LIN {X 0,Y 393.539,Z 325.887,A -85,B 0,C 180,E1 -11593.396,E2 -11593.396} C_VEL
LIN {X 0,Y 392.69,Z 337.53,A -85,B 0,C 180,E1 -11594.293,E2 -11594.293} C_VEL
LIN {X 0,Y 391.726,Z 349.247,A -85,B 0,C 180,E1 -11595.452,E2 -11595.452} C_VEL
LIN {X 0,Y 390.912,Z 359.683,A -85,B 0,C 180,E1 -11596.747,E2 -11596.747} C_VEL
LIN {X 0,Y 390.132,Z 369.641,A -85,B 0,C 180,E1 -11598.306,E2 -11598.306} C_VEL
LIN {X 0,Y 389.491,Z 377.653,A -85,B 0,C 180,E1 -11599.866,E2 -11599.866} C_VEL
LIN {X 0,Y 389.148,Z 383.076,A -85,B 0,C 180,E1 -11601.169,E2 -11601.169} C_VEL
LIN {X 0,Y 388.935,Z 388.388,A -85,B 0,C 180,E1 -11602.732,E2 -11602.732} C_VEL
LIN {X 0,Y 388.746,Z 392.346,A -85,B 0,C 180,E1 -11604.227,E2 -11604.227} C_VEL
LIN {X 0,Y 388.735,Z 395.551,A -85,B 0,C 180,E1 -11605.852,E2 -11605.852} C_VEL
LIN {X 0,Y 388.754,Z 397.047,A -85,B 0,C 180,E1 -11606.89,E2 -11606.89} C_VEL
LIN {X 0,Y 388.841,Z 398.09,A -85,B 0,C 180,E1 -11607.927,E2 -11607.927} C_VEL
LIN {X 0,Y 388.803,Z 398.728,A -85,B 0,C 180,E1 -11608.963,E2 -11608.963} C_VEL
LIN {X 0,Y 388.794,Z 398.973,A -85,B 0,C 180,E1 -11609.999,E2 -11609.999} C_VEL
LIN {X 0,Y 388.793,Z 398.812,A -85,B 0,C 180,E1 -11611.035,E2 -11611.035} C_VEL
LIN {X 0,Y 388.835,Z 398.215,A -85,B 0,C 180,E1 -11612.071,E2 -11612.071} C_VEL
LIN {X 0,Y 388.73,Z 395.815,A -85,B 0,C 180,E1 -11614.146,E2 -11614.146} C_VEL
LIN {X 0,Y 388.74,Z 392.749,A -85,B 0,C 180,E1 -11615.765,E2 -11615.765} C_VEL
LIN {X 0,Y 388.933,Z 388.906,A -85,B 0,C 180,E1 -11617.266,E2 -11617.266} C_VEL
LIN {X 0,Y 389.164,Z 383.8,A -85,B 0,C 180,E1 -11618.829,E2 -11618.829} C_VEL
LIN {X 0,Y 389.572,Z 377.412,A -85,B 0,C 180,E1 -11620.392,E2 -11620.392} C_VEL
LIN {X 0,Y 390.307,Z 369.45,A -85,B 0,C 180,E1 -11621.95,E2 -11621.95} C_VEL
LIN {X 0,Y 390.985,Z 361.36,A -85,B 0,C 180,E1 -11623.248,E2 -11623.248} C_VEL
LIN {X 0,Y 391.894,Z 350.457,A -85,B 0,C 180,E1 -11624.672,E2 -11624.672} C_VEL
LIN {X 0,Y 392.909,Z 339.24,A -85,B 0,C 180,E1 -11625.829,E2 -11625.829} C_VEL
LIN {X 0,Y 393.978,Z 326.812,A -85,B 0,C 180,E1 -11626.831,E2 -11626.831} C_VEL
LIN {X 0,Y 393.281,Z 315.643,A -85,B 0,C 180,E1 -11627.595,E2 -11627.595} C_VEL
LIN {X 0,Y 391.789,Z 303.67,A -85,B 0,C 180,E1 -11628.259,E2 -11628.259} C_VEL
LIN {X 0,Y 389.28,Z 290.364,A -85,B 0,C 180,E1 -11628.842,E2 -11628.842} C_VEL
LIN {X 0,Y 389.711,Z 282.607,A -85,B 0,C 180,E1 -11632.253,E2 -11632.253} C_VEL
LIN {X 0,Y 390.203,Z 274.859,A -85,B 0,C 180,E1 -11635.767,E2 -11635.767} C_VEL
LIN {X 0,Y 390.851,Z 266.706,A -85,B 0,C 180,E1 -11639.635,E2 -11639.635} C_VEL
LIN {X 0,Y 391.527,Z 260.737,A -85,B 0,C 180,E1 -11642.581,E2 -11642.581} C_VEL
LIN {X 0,Y 392.181,Z 254.889,A -85,B 0,C 180,E1 -11645.619,E2 -11645.619} C_VEL
LIN {X 0,Y 392.109,Z 251.439,A -85,B 0,C 180,E1 -11647.545,E2 -11647.545} C_VEL
LIN {X 0,Y 391.372,Z 246.985,A -85,B 0,C 180,E1 -11650.274,E2 -11650.274} C_VEL
LIN {X 0,Y 390.34,Z 241.535,A -85,B 0,C 180,E1 -11653.928,E2 -11653.928} C_VEL
LIN {X 0,Y 390.045,Z 239.9,A -85,B 0,C 180,E1 -11655.167,E2 -11655.167} C_VEL
LIN {X 0,Y 390.03,Z 239.904,A -85,B 0,C 180,E1 -11658.185,E2 -11658.185} C_VEL
LIN {X 0,Y 390.09,Z 239.897,A -85,B 0,C 180,E1 -11660.906,E2 -11660.906} C_VEL
LIN {X 0,Y 390.084,Z 239.897,A -85,B 0,C 180,E1 -11664.792,E2 -11664.792} C_VEL
LIN {X 0,Y 390.021,Z 239.904,A -85,B 0,C 180,E1 -11668.494,E2 -11668.494} C_VEL
LIN {X 0,Y 390.115,Z 239.892,A -85,B 0,C 180,E1 -11672.068,E2 -11672.068} C_VEL
LIN {X 0,Y 390.076,Z 239.898,A -85,B 0,C 180,E1 -11675.518,E2 -11675.518} C_VEL
LIN {X 0,Y 390.052,Z 239.899,A -85,B 0,C 180,E1 -11678.876,E2 -11678.876} C_VEL
LIN {X 0,Y 390.124,Z 239.891,A -85,B 0,C 180,E1 -11682.165,E2 -11682.165} C_VEL
LIN {X 0,Y 390.143,Z 239.888,A -85,B 0,C 180,E1 -11685.391,E2 -11685.391} C_VEL
LIN {X 0,Y 390.154,Z 239.887,A -85,B 0,C 180,E1 -11688.57,E2 -11688.57} C_VEL
LIN {X 0,Y 390.339,Z 239.865,A -85,B 0,C 180,E1 -11691.991,E2 -11691.991} C_VEL
LIN {X 0,Y 390.223,Z 239.879,A -85,B 0,C 180,E1 -11694.832,E2 -11694.832} C_VEL
LIN {X 0,Y 390.415,Z 239.855,A -85,B 0,C 180,E1 -11697.935,E2 -11697.935} C_VEL
LIN {X 0,Y 390.544,Z 239.839,A -85,B 0,C 180,E1 -11699.998,E2 -11699.998} C_VEL
LIN {X 0,Y 390.31,Z 239.869,A -85,B 0,C 180,E1 -11703.095,E2 -11703.095} C_VEL
LIN {X 0,Y 390.302,Z 239.867,A -85,B 0,C 180,E1 -11706.648,E2 -11706.648} C_VEL
LIN {X 0,Y 390.203,Z 239.881,A -85,B 0,C 180,E1 -11709.327,E2 -11709.327} C_VEL
LIN {X 0,Y 390.171,Z 239.886,A -85,B 0,C 180,E1 -11712.481,E2 -11712.481} C_VEL
LIN {X 0,Y 390.121,Z 239.897,A -85,B 0,C 180,E1 -11715.676,E2 -11715.676} C_VEL
LIN {X 0,Y 389.955,Z 239.916,A -85,B 0,C 180,E1 -11717.84,E2 -11717.84} C_VEL
LIN {X 0,Y 389.846,Z 239.927,A -85,B 0,C 180,E1 -11718.933,E2 -11718.933} C_VEL
LIN {X 0,Y 389.827,Z 240.738,A -85,B 0,C 180,E1 -11720.37,E2 -11720.37} C_VEL
LIN {X 0,Y 389.668,Z 243.353,A -85,B 0,C 180,E1 -11723.375,E2 -11723.375} C_VEL
LIN {X 0,Y 389.498,Z 246.382,A -85,B 0,C 180,E1 -11726.812,E2 -11726.812} C_VEL
LIN {X 0,Y 389.338,Z 249.607,A -85,B 0,C 180,E1 -11730.358,E2 -11730.358} C_VEL
LIN {X 0,Y 389.249,Z 252.851,A -85,B 0,C 180,E1 -11733.848,E2 -11733.848} C_VEL
LIN {X 0,Y 389.228,Z 253.251,A -85,B 0,C 180,E1 -11734.27,E2 -11734.27} C_VEL
LIN {X 0,Y 393.317,Z 267.675,A -85,B 0,C 180,E1 -11735.072,E2 -11735.072} C_VEL
LIN {X 0,Y 395.386,Z 276.722,A -85,B 0,C 180,E1 -11735.684,E2 -11735.684} C_VEL
LIN {X 0,Y 395.071,Z 285.643,A -85,B 0,C 180,E1 -11736.275,E2 -11736.275} C_VEL
LIN {X 0,Y 394.145,Z 297.508,A -85,B 0,C 180,E1 -11737.25,E2 -11737.25} C_VEL
LIN {X 0,Y 393.269,Z 308.37,A -85,B 0,C 180,E1 -11738.384,E2 -11738.384} C_VEL
LIN {X 0,Y 392.418,Z 317.961,A -85,B 0,C 180,E1 -11739.638,E2 -11739.638} C_VEL
LIN {X 0,Y 391.501,Z 326.855,A -85,B 0,C 180,E1 -11741.067,E2 -11741.067} C_VEL
LIN {X 0,Y 390.766,Z 334.06,A -85,B 0,C 180,E1 -11742.492,E2 -11742.492} C_VEL
LIN {X 0,Y 390.2,Z 339.898,A -85,B 0,C 180,E1 -11743.91,E2 -11743.91} C_VEL
LIN {X 0,Y 389.589,Z 345.975,A -85,B 0,C 180,E1 -11745.792,E2 -11745.792} C_VEL
LIN {X 0,Y 389.15,Z 350.591,A -85,B 0,C 180,E1 -11747.767,E2 -11747.767} C_VEL
LIN {X 0,Y 388.856,Z 353.204,A -85,B 0,C 180,E1 -11749.411,E2 -11749.411} C_VEL
LIN {X 0,Y 388.717,Z 354.747,A -85,B 0,C 180,E1 -11751.023,E2 -11751.023} C_VEL
LIN {X 0,Y 388.619,Z 355.339,A -85,B 0,C 180,E1 -11752.72,E2 -11752.72} C_VEL
LIN {X 0,Y 388.688,Z 354.729,A -85,B 0,C 180,E1 -11754.649,E2 -11754.649} C_VEL
LIN {X 0,Y 388.799,Z 353.172,A -85,B 0,C 180,E1 -11756.25,E2 -11756.25} C_VEL
LIN {X 0,Y 389.078,Z 350.12,A -85,B 0,C 180,E1 -11758.096,E2 -11758.096} C_VEL
LIN {X 0,Y 389.438,Z 345.459,A -85,B 0,C 180,E1 -11760.019,E2 -11760.019} C_VEL
LIN {X 0,Y 389.902,Z 339.743,A -85,B 0,C 180,E1 -11761.762,E2 -11761.762} C_VEL
LIN {X 0,Y 390.516,Z 332.433,A -85,B 0,C 180,E1 -11763.482,E2 -11763.482} C_VEL
LIN {X 0,Y 391.239,Z 324.18,A -85,B 0,C 180,E1 -11765.031,E2 -11765.031} C_VEL
LIN {X 0,Y 392.019,Z 315.383,A -85,B 0,C 180,E1 -11766.363,E2 -11766.363} C_VEL
LIN {X 0,Y 392.877,Z 304.771,A -85,B 0,C 180,E1 -11767.659,E2 -11767.659} C_VEL
LIN {X 0,Y 393.675,Z 293.882,A -85,B 0,C 180,E1 -11768.727,E2 -11768.727} C_VEL
LIN {X 0,Y 394.413,Z 281.56,A -85,B 0,C 180,E1 -11769.669,E2 -11769.669} C_VEL
LIN {X 0,Y 394.535,Z 274.99,A -85,B 0,C 180,E1 -11770.083,E2 -11770.083} C_VEL
LIN {X 0,Y 391.691,Z 262.166,A -85,B 0,C 180,E1 -11770.853,E2 -11770.853} C_VEL
LIN {X 0,Y 389.137,Z 251.879,A -85,B 0,C 180,E1 -11771.338,E2 -11771.338} C_VEL
LIN {X 0,Y 389.188,Z 248.895,A -85,B 0,C 180,E1 -11774.285,E2 -11774.285} C_VEL
LIN {X 0,Y 389.318,Z 245.691,A -85,B 0,C 180,E1 -11777.49,E2 -11777.49} C_VEL
LIN {X 0,Y 389.404,Z 242.607,A -85,B 0,C 180,E1 -11780.653,E2 -11780.653} C_VEL
LIN {X 0,Y 389.585,Z 240.496,A -85,B 0,C 180,E1 -11782.813,E2 -11782.813} C_VEL
LIN {X 0,Y 389.624,Z 239.954,A -85,B 0,C 180,E1 -11783.788,E2 -11783.788} C_VEL
LIN {X 0,Y 389.784,Z 239.933,A -85,B 0,C 180,E1 -11785.865,E2 -11785.865} C_VEL
LIN {X 0,Y 390.231,Z 239.876,A -85,B 0,C 180,E1 -11787.937,E2 -11787.937} C_VEL
LIN {X 0,Y 390.533,Z 239.838,A -85,B 0,C 180,E1 -11790.001,E2 -11790.001} C_VEL
LIN {X 0,Y 390.303,Z 239.869,A -85,B 0,C 180,E1 -11793.098,E2 -11793.098} C_VEL
LIN {X 0,Y 390.316,Z 239.864,A -85,B 0,C 180,E1 -11796.203,E2 -11796.203} C_VEL
LIN {X 0,Y 390.301,Z 239.866,A -85,B 0,C 180,E1 -11798.283,E2 -11798.283} C_VEL
LIN {X 0,Y 390.167,Z 239.883,A -85,B 0,C 180,E1 -11802.484,E2 -11802.484} C_VEL
LIN {X 0,Y 390.111,Z 239.889,A -85,B 0,C 180,E1 -11806.087,E2 -11806.087} C_VEL
LIN {X 0,Y 389.448,Z 239.976,A -85,B 0,C 180,E1 -11806.949,E2 -11806.949} C_VEL
LIN {X 0,Y 386.62,Z 240.325,A -85,B 0,C 180,E1 -11808.349,E2 -11808.349} C_VEL
LIN {X 0,Y 384.208,Z 240.627,A -85,B 0,C 180,E1 -11809.481,E2 -11809.481} C_VEL
LIN {X 0,Y 383.148,Z 240.758,A -85,B 0,C 180,E1 -11810.356,E2 -11810.356} C_VEL
LIN {X 0,Y 383.048,Z 240.772,A -85,B 0,C 180,E1 -11810.652,E2 -11810.652} C_VEL
LIN {X 0,Y 383.031,Z 240.771,A -85,B 0,C 180,E1 -11813.809,E2 -11813.809} C_VEL
LIN {X 0,Y 383.046,Z 240.772,A -85,B 0,C 180,E1 -11817.304,E2 -11817.304} C_VEL
LIN {X 0,Y 382.973,Z 240.783,A -85,B 0,C 180,E1 -11820.921,E2 -11820.921} C_VEL
LIN {X 0,Y 383.01,Z 240.778,A -85,B 0,C 180,E1 -11824.67,E2 -11824.67} C_VEL
LIN {X 0,Y 382.996,Z 240.775,A -85,B 0,C 180,E1 -11827.907,E2 -11827.907} C_VEL
LIN {X 0,Y 383.04,Z 240.771,A -85,B 0,C 180,E1 -11831.341,E2 -11831.341} C_VEL
LIN {X 0,Y 383.028,Z 240.775,A -85,B 0,C 180,E1 -11834.311,E2 -11834.311} C_VEL
LIN {X 0,Y 383.035,Z 240.771,A -85,B 0,C 180,E1 -11837.246,E2 -11837.246} C_VEL
LIN {X 0,Y 383.018,Z 240.777,A -85,B 0,C 180,E1 -11840.414,E2 -11840.414} C_VEL
LIN {X 0,Y 383.024,Z 240.775,A -85,B 0,C 180,E1 -11844.047,E2 -11844.047} C_VEL
LIN {X 0,Y 382.985,Z 240.777,A -85,B 0,C 180,E1 -11847.58,E2 -11847.58} C_VEL
LIN {X 0,Y 382.991,Z 240.781,A -85,B 0,C 180,E1 -11850.302,E2 -11850.302} C_VEL
LIN {X 0,Y 383.08,Z 240.769,A -85,B 0,C 180,E1 -11854.023,E2 -11854.023} C_VEL
LIN {X 0,Y 383.009,Z 240.774,A -85,B 0,C 180,E1 -11857.337,E2 -11857.337} C_VEL
LIN {X 0,Y 383.063,Z 240.768,A -85,B 0,C 180,E1 -11860.718,E2 -11860.718} C_VEL
LIN {X 0,Y 383.085,Z 240.769,A -85,B 0,C 180,E1 -11864.029,E2 -11864.029} C_VEL
LIN {X 0,Y 383.145,Z 240.757,A -85,B 0,C 180,E1 -11867.286,E2 -11867.286} C_VEL
LIN {X 0,Y 383.15,Z 240.758,A -85,B 0,C 180,E1 -11870.5,E2 -11870.5} C_VEL
LIN {X 0,Y 383.279,Z 240.744,A -85,B 0,C 180,E1 -11873.685,E2 -11873.685} C_VEL
LIN {X 0,Y 383.391,Z 240.73,A -85,B 0,C 180,E1 -11877.901,E2 -11877.901} C_VEL
LIN {X 0,Y 383.524,Z 240.713,A -85,B 0,C 180,E1 -11880.002,E2 -11880.002} C_VEL
LIN {X 0,Y 383.246,Z 240.745,A -85,B 0,C 180,E1 -11883.155,E2 -11883.155} C_VEL
LIN {X 0,Y 383.279,Z 240.741,A -85,B 0,C 180,E1 -11886.318,E2 -11886.318} C_VEL
LIN {X 0,Y 383.151,Z 240.761,A -85,B 0,C 180,E1 -11889.504,E2 -11889.504} C_VEL
LIN {X 0,Y 383.134,Z 240.763,A -85,B 0,C 180,E1 -11893.537,E2 -11893.537} C_VEL
LIN {X 0,Y 383.104,Z 240.766,A -85,B 0,C 180,E1 -11897.455,E2 -11897.455} C_VEL
LIN {X 0,Y 383.038,Z 240.771,A -85,B 0,C 180,E1 -11900.648,E2 -11900.648} C_VEL
LIN {X 0,Y 383.042,Z 240.772,A -85,B 0,C 180,E1 -11903.808,E2 -11903.808} C_VEL
LIN {X 0,Y 383.089,Z 240.764,A -85,B 0,C 180,E1 -11906.124,E2 -11906.124} C_VEL
LIN {X 0,Y 383.002,Z 240.776,A -85,B 0,C 180,E1 -11909.7,E2 -11909.7} C_VEL
LIN {X 0,Y 383.013,Z 240.777,A -85,B 0,C 180,E1 -11913.401,E2 -11913.401} C_VEL
LIN {X 0,Y 383.041,Z 240.77,A -85,B 0,C 180,E1 -11916.165,E2 -11916.165} C_VEL
LIN {X 0,Y 383.017,Z 240.777,A -85,B 0,C 180,E1 -11919.959,E2 -11919.959} C_VEL
LIN {X 0,Y 383.015,Z 240.777,A -85,B 0,C 180,E1 -11922.779,E2 -11922.779} C_VEL
LIN {X 0,Y 383.041,Z 240.901,A -85,B 0,C 180,E1 -11926.17,E2 -11926.17} C_VEL
LIN {X 0,Y 384.068,Z 246.503,A -85,B 0,C 180,E1 -11929.487,E2 -11929.487} C_VEL
LIN {X 0,Y 385.047,Z 252.722,A -85,B 0,C 180,E1 -11932.962,E2 -11932.962} C_VEL
LIN {X 0,Y 384.98,Z 257.096,A -85,B 0,C 180,E1 -11935.237,E2 -11935.237} C_VEL
LIN {X 0,Y 384.2,Z 263.851,A -85,B 0,C 180,E1 -11938.577,E2 -11938.577} C_VEL
LIN {X 0,Y 383.515,Z 271.311,A -85,B 0,C 180,E1 -11942.155,E2 -11942.155} C_VEL
LIN {X 0,Y 382.938,Z 278.749,A -85,B 0,C 180,E1 -11945.609,E2 -11945.609} C_VEL
LIN {X 0,Y 382.451,Z 286.173,A -85,B 0,C 180,E1 -11949.001,E2 -11949.001} C_VEL
LIN {X 0,Y 382.199,Z 291.545,A -85,B 0,C 180,E1 -11951.332,E2 -11951.332} C_VEL
LIN {X 0,Y 384.466,Z 305.306,A -85,B 0,C 180,E1 -11951.894,E2 -11951.894} C_VEL
LIN {X 0,Y 385.992,Z 318.448,A -85,B 0,C 180,E1 -11952.637,E2 -11952.637} C_VEL
LIN {X 0,Y 386.586,Z 326.938,A -85,B 0,C 180,E1 -11953.225,E2 -11953.225} C_VEL
LIN {X 0,Y 385.704,Z 338.233,A -85,B 0,C 180,E1 -11954.137,E2 -11954.137} C_VEL
LIN {X 0,Y 384.733,Z 349.624,A -85,B 0,C 180,E1 -11955.301,E2 -11955.301} C_VEL
LIN {X 0,Y 383.975,Z 359.086,A -85,B 0,C 180,E1 -11956.504,E2 -11956.504} C_VEL
LIN {X 0,Y 383.253,Z 367.589,A -85,B 0,C 180,E1 -11957.825,E2 -11957.825} C_VEL
LIN {X 0,Y 382.494,Z 375.884,A -85,B 0,C 180,E1 -11959.411,E2 -11959.411} C_VEL
LIN {X 0,Y 382.067,Z 382.577,A -85,B 0,C 180,E1 -11961.004,E2 -11961.004} C_VEL
LIN {X 0,Y 381.858,Z 387.913,A -85,B 0,C 180,E1 -11962.597,E2 -11962.597} C_VEL
LIN {X 0,Y 381.682,Z 391.361,A -85,B 0,C 180,E1 -11963.896,E2 -11963.896} C_VEL
LIN {X 0,Y 381.661,Z 395.113,A -85,B 0,C 180,E1 -11965.775,E2 -11965.775} C_VEL
LIN {X 0,Y 381.657,Z 396.621,A -85,B 0,C 180,E1 -11966.832,E2 -11966.832} C_VEL
LIN {X 0,Y 381.754,Z 397.674,A -85,B 0,C 180,E1 -11967.889,E2 -11967.889} C_VEL
LIN {X 0,Y 381.733,Z 398.319,A -85,B 0,C 180,E1 -11968.944,E2 -11968.944} C_VEL
LIN {X 0,Y 381.721,Z 398.571,A -85,B 0,C 180,E1 -11969.999,E2 -11969.999} C_VEL
LIN {X 0,Y 381.724,Z 398.421,A -85,B 0,C 180,E1 -11971.054,E2 -11971.054} C_VEL
LIN {X 0,Y 381.747,Z 397.831,A -85,B 0,C 180,E1 -11972.109,E2 -11972.109} C_VEL
LIN {X 0,Y 381.654,Z 395.445,A -85,B 0,C 180,E1 -11974.223,E2 -11974.223} C_VEL
LIN {X 0,Y 381.695,Z 391.851,A -85,B 0,C 180,E1 -11976.122,E2 -11976.122} C_VEL
LIN {X 0,Y 381.906,Z 387.001,A -85,B 0,C 180,E1 -11977.932,E2 -11977.932} C_VEL
LIN {X 0,Y 382.289,Z 380.466,A -85,B 0,C 180,E1 -11979.79,E2 -11979.79} C_VEL
LIN {X 0,Y 382.859,Z 373.368,A -85,B 0,C 180,E1 -11981.38,E2 -11981.38} C_VEL
LIN {X 0,Y 383.809,Z 364.519,A -85,B 0,C 180,E1 -11982.961,E2 -11982.961} C_VEL
LIN {X 0,Y 384.627,Z 354.374,A -85,B 0,C 180,E1 -11984.432,E2 -11984.432} C_VEL
LIN {X 0,Y 385.581,Z 344.377,A -85,B 0,C 180,E1 -11985.595,E2 -11985.595} C_VEL
LIN {X 0,Y 386.658,Z 333.213,A -85,B 0,C 180,E1 -11986.634,E2 -11986.634} C_VEL
LIN {X 0,Y 387.076,Z 325.209,A -85,B 0,C 180,E1 -11987.261,E2 -11987.261} C_VEL
LIN {X 0,Y 386.267,Z 314.248,A -85,B 0,C 180,E1 -11988.016,E2 -11988.016} C_VEL
LIN {X 0,Y 384.573,Z 302.084,A -85,B 0,C 180,E1 -11988.7,E2 -11988.7} C_VEL
LIN {X 0,Y 382.278,Z 289.943,A -85,B 0,C 180,E1 -11989.249,E2 -11989.249} C_VEL
LIN {X 0,Y 382.678,Z 282.313,A -85,B 0,C 180,E1 -11992.684,E2 -11992.684} C_VEL
LIN {X 0,Y 383.198,Z 274.95,A -85,B 0,C 180,E1 -11996.113,E2 -11996.113} C_VEL
LIN {X 0,Y 383.904,Z 266.636,A -85,B 0,C 180,E1 -12000.15,E2 -12000.15} C_VEL
LIN {X 0,Y 384.669,Z 260.569,A -85,B 0,C 180,E1 -12003.236,E2 -12003.236} C_VEL
LIN {X 0,Y 385.21,Z 255.953,A -85,B 0,C 180,E1 -12005.719,E2 -12005.719} C_VEL
LIN {X 0,Y 385.106,Z 252.584,A -85,B 0,C 180,E1 -12007.638,E2 -12007.638} C_VEL
LIN {X 0,Y 384.341,Z 248.06,A -85,B 0,C 180,E1 -12010.475,E2 -12010.475} C_VEL
LIN {X 0,Y 383.295,Z 242.437,A -85,B 0,C 180,E1 -12014.348,E2 -12014.348} C_VEL
LIN {X 0,Y 382.995,Z 240.78,A -85,B 0,C 180,E1 -12015.695,E2 -12015.695} C_VEL
LIN {X 0,Y 382.987,Z 240.781,A -85,B 0,C 180,E1 -12018.794,E2 -12018.794} C_VEL
LIN {X 0,Y 383,Z 240.78,A -85,B 0,C 180,E1 -12022.094,E2 -12022.094} C_VEL
LIN {X 0,Y 383.017,Z 240.778,A -85,B 0,C 180,E1 -12025.331,E2 -12025.331} C_VEL
LIN {X 0,Y 382.981,Z 240.783,A -85,B 0,C 180,E1 -12029.08,E2 -12029.08} C_VEL
LIN {X 0,Y 383.054,Z 240.772,A -85,B 0,C 180,E1 -12032.696,E2 -12032.696} C_VEL
LIN {X 0,Y 383.049,Z 240.773,A -85,B 0,C 180,E1 -12035.038,E2 -12035.038} C_VEL
LIN {X 0,Y 382.99,Z 240.779,A -85,B 0,C 180,E1 -12038.467,E2 -12038.467} C_VEL
LIN {X 0,Y 383.086,Z 240.768,A -85,B 0,C 180,E1 -12041.826,E2 -12041.826} C_VEL
LIN {X 0,Y 383.108,Z 240.765,A -85,B 0,C 180,E1 -12045.117,E2 -12045.117} C_VEL
LIN {X 0,Y 383.103,Z 240.766,A -85,B 0,C 180,E1 -12048.357,E2 -12048.357} C_VEL
LIN {X 0,Y 383.299,Z 240.742,A -85,B 0,C 180,E1 -12051.931,E2 -12051.931} C_VEL
LIN {X 0,Y 383.195,Z 240.754,A -85,B 0,C 180,E1 -12054.737,E2 -12054.737} C_VEL
LIN {X 0,Y 383.382,Z 240.731,A -85,B 0,C 180,E1 -12057.897,E2 -12057.897} C_VEL
LIN {X 0,Y 383.513,Z 240.715,A -85,B 0,C 180,E1 -12059.998,E2 -12059.998} C_VEL
LIN {X 0,Y 383.246,Z 240.748,A -85,B 0,C 180,E1 -12063.152,E2 -12063.152} C_VEL
LIN {X 0,Y 383.261,Z 240.745,A -85,B 0,C 180,E1 -12066.642,E2 -12066.642} C_VEL
LIN {X 0,Y 383.252,Z 240.748,A -85,B 0,C 180,E1 -12068.434,E2 -12068.434} C_VEL
LIN {X 0,Y 383.102,Z 240.766,A -85,B 0,C 180,E1 -12071.64,E2 -12071.64} C_VEL
LIN {X 0,Y 383.1,Z 240.77,A -85,B 0,C 180,E1 -12074.88,E2 -12074.88} C_VEL
LIN {X 0,Y 382.989,Z 240.785,A -85,B 0,C 180,E1 -12077.408,E2 -12077.408} C_VEL
LIN {X 0,Y 382.769,Z 240.862,A -85,B 0,C 180,E1 -12079.297,E2 -12079.297} C_VEL
LIN {X 0,Y 382.723,Z 242.713,A -85,B 0,C 180,E1 -12081.545,E2 -12081.545} C_VEL
LIN {X 0,Y 382.557,Z 245.702,A -85,B 0,C 180,E1 -12084.993,E2 -12084.993} C_VEL
LIN {X 0,Y 382.354,Z 248.841,A -85,B 0,C 180,E1 -12088.546,E2 -12088.546} C_VEL
LIN {X 0,Y 382.251,Z 252.227,A -85,B 0,C 180,E1 -12092.25,E2 -12092.25} C_VEL
LIN {X 0,Y 382.201,Z 253.728,A -85,B 0,C 180,E1 -12093.882,E2 -12093.882} C_VEL
LIN {X 0,Y 386.087,Z 266.944,A -85,B 0,C 180,E1 -12094.628,E2 -12094.628} C_VEL
LIN {X 0,Y 388.789,Z 279.097,A -85,B 0,C 180,E1 -12095.468,E2 -12095.468} C_VEL
LIN {X 0,Y 387.975,Z 291.331,A -85,B 0,C 180,E1 -12096.353,E2 -12096.353} C_VEL
LIN {X 0,Y 386.984,Z 302.616,A -85,B 0,C 180,E1 -12097.402,E2 -12097.402} C_VEL
LIN {X 0,Y 386.148,Z 312.086,A -85,B 0,C 180,E1 -12098.501,E2 -12098.501} C_VEL
LIN {X 0,Y 385.359,Z 320.346,A -85,B 0,C 180,E1 -12099.663,E2 -12099.663} C_VEL
LIN {X 0,Y 384.374,Z 329.115,A -85,B 0,C 180,E1 -12101.162,E2 -12101.162} C_VEL
LIN {X 0,Y 383.552,Z 337.022,A -85,B 0,C 180,E1 -12102.868,E2 -12102.868} C_VEL
LIN {X 0,Y 382.875,Z 343.552,A -85,B 0,C 180,E1 -12104.662,E2 -12104.662} C_VEL
LIN {X 0,Y 382.378,Z 348.466,A -85,B 0,C 180,E1 -12106.451,E2 -12106.451} C_VEL
LIN {X 0,Y 382.045,Z 351.54,A -85,B 0,C 180,E1 -12107.933,E2 -12107.933} C_VEL
LIN {X 0,Y 381.731,Z 354.243,A -85,B 0,C 180,E1 -12109.882,E2 -12109.882} C_VEL
LIN {X 0,Y 381.613,Z 355.332,A -85,B 0,C 180,E1 -12111.234,E2 -12111.234} C_VEL
LIN {X 0,Y 381.561,Z 355.726,A -85,B 0,C 180,E1 -12112.569,E2 -12112.569} C_VEL
LIN {X 0,Y 381.565,Z 355.405,A -85,B 0,C 180,E1 -12114.134,E2 -12114.134} C_VEL
LIN {X 0,Y 381.696,Z 353.944,A -85,B 0,C 180,E1 -12115.947,E2 -12115.947} C_VEL
LIN {X 0,Y 381.953,Z 351.182,A -85,B 0,C 180,E1 -12117.819,E2 -12117.819} C_VEL
LIN {X 0,Y 382.296,Z 346.802,A -85,B 0,C 180,E1 -12119.768,E2 -12119.768} C_VEL
LIN {X 0,Y 382.721,Z 341.574,A -85,B 0,C 180,E1 -12121.483,E2 -12121.483} C_VEL
LIN {X 0,Y 383.412,Z 334.342,A -85,B 0,C 180,E1 -12123.317,E2 -12123.317} C_VEL
LIN {X 0,Y 384.078,Z 326.806,A -85,B 0,C 180,E1 -12124.823,E2 -12124.823} C_VEL
LIN {X 0,Y 384.933,Z 317.553,A -85,B 0,C 180,E1 -12126.319,E2 -12126.319} C_VEL
LIN {X 0,Y 385.714,Z 308.555,A -85,B 0,C 180,E1 -12127.504,E2 -12127.504} C_VEL
LIN {X 0,Y 386.558,Z 297.547,A -85,B 0,C 180,E1 -12128.679,E2 -12128.679} C_VEL
LIN {X 0,Y 387.392,Z 285.33,A -85,B 0,C 180,E1 -12129.7,E2 -12129.7} C_VEL
LIN {X 0,Y 387.783,Z 276.739,A -85,B 0,C 180,E1 -12130.273,E2 -12130.273} C_VEL
LIN {X 0,Y 384.841,Z 263.178,A -85,B 0,C 180,E1 -12131.122,E2 -12131.122} C_VEL
LIN {X 0,Y 382.048,Z 252.228,A -85,B 0,C 180,E1 -12131.674,E2 -12131.674} C_VEL
LIN {X 0,Y 382.126,Z 248.817,A -85,B 0,C 180,E1 -12135.08,E2 -12135.08} C_VEL
LIN {X 0,Y 382.276,Z 245.626,A -85,B 0,C 180,E1 -12138.334,E2 -12138.334} C_VEL
LIN {X 0,Y 382.423,Z 242.507,A -85,B 0,C 180,E1 -12141.547,E2 -12141.547} C_VEL
LIN {X 0,Y 382.524,Z 241.318,A -85,B 0,C 180,E1 -12142.786,E2 -12142.786} C_VEL
LIN {X 0,Y 382.56,Z 240.835,A -85,B 0,C 180,E1 -12143.673,E2 -12143.673} C_VEL
LIN {X 0,Y 382.742,Z 240.811,A -85,B 0,C 180,E1 -12145.789,E2 -12145.789} C_VEL
LIN {X 0,Y 383.284,Z 240.742,A -85,B 0,C 180,E1 -12148.95,E2 -12148.95} C_VEL
LIN {X 0,Y 383.502,Z 240.713,A -85,B 0,C 180,E1 -12150.001,E2 -12150.001} C_VEL
LIN {X 0,Y 383.24,Z 240.75,A -85,B 0,C 180,E1 -12153.155,E2 -12153.155} C_VEL
LIN {X 0,Y 383.273,Z 240.741,A -85,B 0,C 180,E1 -12156.318,E2 -12156.318} C_VEL
LIN {X 0,Y 383.247,Z 240.744,A -85,B 0,C 180,E1 -12158.437,E2 -12158.437} C_VEL
LIN {X 0,Y 383.097,Z 240.765,A -85,B 0,C 180,E1 -12161.643,E2 -12161.643} C_VEL
LIN {X 0,Y 383.1,Z 240.767,A -85,B 0,C 180,E1 -12164.883,E2 -12164.883} C_VEL
LIN {X 0,Y 383.082,Z 240.765,A -85,B 0,C 180,E1 -12168.174,E2 -12168.174} C_VEL
LIN {X 0,Y 383.048,Z 240.772,A -85,B 0,C 180,E1 -12170.652,E2 -12170.652} C_VEL
LIN {X 0,Y 382.336,Z 240.866,A -85,B 0,C 180,E1 -12171.531,E2 -12171.531} C_VEL
LIN {X 0,Y 379.448,Z 241.222,A -85,B 0,C 180,E1 -12172.958,E2 -12172.958} C_VEL
LIN {X 0,Y 377.048,Z 241.516,A -85,B 0,C 180,E1 -12174.112,E2 -12174.112} C_VEL
LIN {X 0,Y 376.051,Z 241.645,A -85,B 0,C 180,E1 -12175.005,E2 -12175.005} C_VEL
LIN {X 0,Y 375.986,Z 241.649,A -85,B 0,C 180,E1 -12175.307,E2 -12175.307} C_VEL
LIN {X 0,Y 375.99,Z 241.651,A -85,B 0,C 180,E1 -12178.54,E2 -12178.54} C_VEL
LIN {X 0,Y 375.948,Z 241.654,A -85,B 0,C 180,E1 -12181.564,E2 -12181.564} C_VEL
LIN {X 0,Y 375.95,Z 241.654,A -85,B 0,C 180,E1 -12185.418,E2 -12185.418} C_VEL
LIN {X 0,Y 375.971,Z 241.652,A -85,B 0,C 180,E1 -12188.273,E2 -12188.273} C_VEL
LIN {X 0,Y 375.983,Z 241.649,A -85,B 0,C 180,E1 -12191.612,E2 -12191.612} C_VEL
LIN {X 0,Y 375.963,Z 241.652,A -85,B 0,C 180,E1 -12195.264,E2 -12195.264} C_VEL
LIN {X 0,Y 375.977,Z 241.65,A -85,B 0,C 180,E1 -12199.141,E2 -12199.141} C_VEL
LIN {X 0,Y 375.965,Z 241.652,A -85,B 0,C 180,E1 -12201.914,E2 -12201.914} C_VEL
LIN {X 0,Y 375.978,Z 241.65,A -85,B 0,C 180,E1 -12205.335,E2 -12205.335} C_VEL
LIN {X 0,Y 375.956,Z 241.657,A -85,B 0,C 180,E1 -12208.44,E2 -12208.44} C_VEL
LIN {X 0,Y 375.983,Z 241.653,A -85,B 0,C 180,E1 -12212.143,E2 -12212.143} C_VEL
LIN {X 0,Y 376.007,Z 241.649,A -85,B 0,C 180,E1 -12214.541,E2 -12214.541} C_VEL
LIN {X 0,Y 375.964,Z 241.656,A -85,B 0,C 180,E1 -12218.048,E2 -12218.048} C_VEL
LIN {X 0,Y 376.027,Z 241.644,A -85,B 0,C 180,E1 -12221.476,E2 -12221.476} C_VEL
LIN {X 0,Y 376.063,Z 241.639,A -85,B 0,C 180,E1 -12224.835,E2 -12224.835} C_VEL
LIN {X 0,Y 376.063,Z 241.643,A -85,B 0,C 180,E1 -12228.139,E2 -12228.139} C_VEL
LIN {X 0,Y 376.205,Z 241.626,A -85,B 0,C 180,E1 -12231.941,E2 -12231.941} C_VEL
LIN {X 0,Y 376.173,Z 241.625,A -85,B 0,C 180,E1 -12234.642,E2 -12234.642} C_VEL
LIN {X 0,Y 376.357,Z 241.607,A -85,B 0,C 180,E1 -12237.861,E2 -12237.861} C_VEL
LIN {X 0,Y 376.494,Z 241.589,A -85,B 0,C 180,E1 -12240.002,E2 -12240.002} C_VEL
LIN {X 0,Y 376.357,Z 241.604,A -85,B 0,C 180,E1 -12242.142,E2 -12242.142} C_VEL
LIN {X 0,Y 376.236,Z 241.618,A -85,B 0,C 180,E1 -12246.437,E2 -12246.437} C_VEL
LIN {X 0,Y 376.121,Z 241.636,A -85,B 0,C 180,E1 -12249.683,E2 -12249.683} C_VEL
LIN {X 0,Y 376.098,Z 241.639,A -85,B 0,C 180,E1 -12253.659,E2 -12253.659} C_VEL
LIN {X 0,Y 376.052,Z 241.645,A -85,B 0,C 180,E1 -12257.608,E2 -12257.608} C_VEL
LIN {X 0,Y 375.988,Z 241.65,A -85,B 0,C 180,E1 -12260.833,E2 -12260.833} C_VEL
LIN {X 0,Y 376.002,Z 241.646,A -85,B 0,C 180,E1 -12264.282,E2 -12264.282} C_VEL
LIN {X 0,Y 376.029,Z 241.644,A -85,B 0,C 180,E1 -12266.653,E2 -12266.653} C_VEL
LIN {X 0,Y 375.974,Z 241.65,A -85,B 0,C 180,E1 -12270.313,E2 -12270.313} C_VEL
LIN {X 0,Y 375.97,Z 241.651,A -85,B 0,C 180,E1 -12274.112,E2 -12274.112} C_VEL
LIN {X 0,Y 375.962,Z 241.654,A -85,B 0,C 180,E1 -12276.742,E2 -12276.742} C_VEL
LIN {X 0,Y 375.997,Z 241.652,A -85,B 0,C 180,E1 -12279.971,E2 -12279.971} C_VEL
LIN {X 0,Y 375.939,Z 241.657,A -85,B 0,C 180,E1 -12283.766,E2 -12283.766} C_VEL
LIN {X 0,Y 376,Z 241.814,A -85,B 0,C 180,E1 -12285.896,E2 -12285.896} C_VEL
LIN {X 0,Y 377.015,Z 247.396,A -85,B 0,C 180,E1 -12289.273,E2 -12289.273} C_VEL
LIN {X 0,Y 377.839,Z 252.373,A -85,B 0,C 180,E1 -12292.133,E2 -12292.133} C_VEL
LIN {X 0,Y 378.082,Z 256.116,A -85,B 0,C 180,E1 -12294.158,E2 -12294.158} C_VEL
LIN {X 0,Y 377.578,Z 261.41,A -85,B 0,C 180,E1 -12296.889,E2 -12296.889} C_VEL
LIN {X 0,Y 376.801,Z 268.454,A -85,B 0,C 180,E1 -12300.377,E2 -12300.377} C_VEL
LIN {X 0,Y 376.167,Z 275.413,A -85,B 0,C 180,E1 -12303.742,E2 -12303.742} C_VEL
LIN {X 0,Y 375.595,Z 283.28,A -85,B 0,C 180,E1 -12307.443,E2 -12307.443} C_VEL
LIN {X 0,Y 375.166,Z 290.952,A -85,B 0,C 180,E1 -12310.968,E2 -12310.968} C_VEL
LIN {X 0,Y 377.687,Z 306.939,A -85,B 0,C 180,E1 -12311.685,E2 -12311.685} C_VEL
LIN {X 0,Y 379.118,Z 319.5,A -85,B 0,C 180,E1 -12312.435,E2 -12312.435} C_VEL
LIN {X 0,Y 379.633,Z 327.878,A -85,B 0,C 180,E1 -12313.047,E2 -12313.047} C_VEL
LIN {X 0,Y 378.717,Z 338.918,A -85,B 0,C 180,E1 -12313.975,E2 -12313.975} C_VEL
LIN {X 0,Y 377.749,Z 349.699,A -85,B 0,C 180,E1 -12315.111,E2 -12315.111} C_VEL
LIN {X 0,Y 377.036,Z 358.46,A -85,B 0,C 180,E1 -12316.25,E2 -12316.25} C_VEL
LIN {X 0,Y 376.278,Z 367.014,A -85,B 0,C 180,E1 -12317.596,E2 -12317.596} C_VEL
LIN {X 0,Y 375.474,Z 375.34,A -85,B 0,C 180,E1 -12319.211,E2 -12319.211} C_VEL
LIN {X 0,Y 375.007,Z 382.059,A -85,B 0,C 180,E1 -12320.833,E2 -12320.833} C_VEL
LIN {X 0,Y 374.768,Z 387.419,A -85,B 0,C 180,E1 -12322.456,E2 -12322.456} C_VEL
LIN {X 0,Y 374.602,Z 391.201,A -85,B 0,C 180,E1 -12323.913,E2 -12323.913} C_VEL
LIN {X 0,Y 374.586,Z 394.665,A -85,B 0,C 180,E1 -12325.695,E2 -12325.695} C_VEL
LIN {X 0,Y 374.564,Z 396.186,A -85,B 0,C 180,E1 -12326.772,E2 -12326.772} C_VEL
LIN {X 0,Y 374.669,Z 397.253,A -85,B 0,C 180,E1 -12327.849,E2 -12327.849} C_VEL
LIN {X 0,Y 374.665,Z 397.907,A -85,B 0,C 180,E1 -12328.924,E2 -12328.924} C_VEL
LIN {X 0,Y 374.651,Z 398.167,A -85,B 0,C 180,E1 -12329.999,E2 -12329.999} C_VEL
LIN {X 0,Y 374.656,Z 398.029,A -85,B 0,C 180,E1 -12331.074,E2 -12331.074} C_VEL
LIN {X 0,Y 374.646,Z 397.449,A -85,B 0,C 180,E1 -12332.149,E2 -12332.149} C_VEL
LIN {X 0,Y 374.578,Z 395.078,A -85,B 0,C 180,E1 -12334.303,E2 -12334.303} C_VEL
LIN {X 0,Y 374.593,Z 391.859,A -85,B 0,C 180,E1 -12336.074,E2 -12336.074} C_VEL
LIN {X 0,Y 374.766,Z 388.231,A -85,B 0,C 180,E1 -12337.542,E2 -12337.542} C_VEL
LIN {X 0,Y 375.039,Z 383.158,A -85,B 0,C 180,E1 -12339.164,E2 -12339.164} C_VEL
LIN {X 0,Y 375.501,Z 376.807,A -85,B 0,C 180,E1 -12340.786,E2 -12340.786} C_VEL
LIN {X 0,Y 376.342,Z 368.917,A -85,B 0,C 180,E1 -12342.4,E2 -12342.4} C_VEL
LIN {X 0,Y 377.298,Z 359.104,A -85,B 0,C 180,E1 -12344.013,E2 -12344.013} C_VEL
LIN {X 0,Y 378.251,Z 349.004,A -85,B 0,C 180,E1 -12345.352,E2 -12345.352} C_VEL
LIN {X 0,Y 379.407,Z 337.638,A -85,B 0,C 180,E1 -12346.546,E2 -12346.546} C_VEL
LIN {X 0,Y 380.263,Z 328.5,A -85,B 0,C 180,E1 -12347.324,E2 -12347.324} C_VEL
LIN {X 0,Y 379.608,Z 316.421,A -85,B 0,C 180,E1 -12348.221,E2 -12348.221} C_VEL
LIN {X 0,Y 378.023,Z 304.095,A -85,B 0,C 180,E1 -12348.971,E2 -12348.971} C_VEL
LIN {X 0,Y 375.458,Z 290.992,A -85,B 0,C 180,E1 -12349.599,E2 -12349.599} C_VEL
LIN {X 0,Y 375.248,Z 289.507,A -85,B 0,C 180,E1 -12349.66,E2 -12349.66} C_VEL
LIN {X 0,Y 375.66,Z 282.021,A -85,B 0,C 180,E1 -12353.132,E2 -12353.132} C_VEL
LIN {X 0,Y 376.22,Z 274.694,A -85,B 0,C 180,E1 -12356.636,E2 -12356.636} C_VEL
LIN {X 0,Y 376.876,Z 267.484,A -85,B 0,C 180,E1 -12360.23,E2 -12360.23} C_VEL
LIN {X 0,Y 377.825,Z 260.42,A -85,B 0,C 180,E1 -12363.919,E2 -12363.919} C_VEL
LIN {X 0,Y 378.235,Z 255.793,A -85,B 0,C 180,E1 -12366.482,E2 -12366.482} C_VEL
LIN {X 0,Y 377.891,Z 252.278,A -85,B 0,C 180,E1 -12368.636,E2 -12368.636} C_VEL
LIN {X 0,Y 376.999,Z 247.509,A -85,B 0,C 180,E1 -12371.781,E2 -12371.781} C_VEL
LIN {X 0,Y 376.161,Z 242.763,A -85,B 0,C 180,E1 -12375.231,E2 -12375.231} C_VEL
LIN {X 0,Y 375.929,Z 241.661,A -85,B 0,C 180,E1 -12376.232,E2 -12376.232} C_VEL
LIN {X 0,Y 375.988,Z 241.653,A -85,B 0,C 180,E1 -12380.028,E2 -12380.028} C_VEL
LIN {X 0,Y 375.963,Z 241.658,A -85,B 0,C 180,E1 -12383.494,E2 -12383.494} C_VEL
LIN {X 0,Y 375.958,Z 241.657,A -85,B 0,C 180,E1 -12385.887,E2 -12385.887} C_VEL
LIN {X 0,Y 375.962,Z 241.655,A -85,B 0,C 180,E1 -12389.686,E2 -12389.686} C_VEL
LIN {X 0,Y 376.017,Z 241.648,A -85,B 0,C 180,E1 -12393.346,E2 -12393.346} C_VEL
LIN {X 0,Y 375.993,Z 241.652,A -85,B 0,C 180,E1 -12396.887,E2 -12396.887} C_VEL
LIN {X 0,Y 375.994,Z 241.651,A -85,B 0,C 180,E1 -12400.338,E2 -12400.338} C_VEL
LIN {X 0,Y 376.025,Z 241.648,A -85,B 0,C 180,E1 -12403.717,E2 -12403.717} C_VEL
LIN {X 0,Y 376.102,Z 241.638,A -85,B 0,C 180,E1 -12407.04,E2 -12407.04} C_VEL
LIN {X 0,Y 376.119,Z 241.635,A -85,B 0,C 180,E1 -12410.317,E2 -12410.317} C_VEL
LIN {X 0,Y 376.225,Z 241.623,A -85,B 0,C 180,E1 -12412.485,E2 -12412.485} C_VEL
LIN {X 0,Y 376.167,Z 241.629,A -85,B 0,C 180,E1 -12414.638,E2 -12414.638} C_VEL
LIN {X 0,Y 376.348,Z 241.607,A -85,B 0,C 180,E1 -12417.858,E2 -12417.858} C_VEL
LIN {X 0,Y 376.482,Z 241.59,A -85,B 0,C 180,E1 -12419.998,E2 -12419.998} C_VEL
LIN {X 0,Y 376.184,Z 241.628,A -85,B 0,C 180,E1 -12423.211,E2 -12423.211} C_VEL
LIN {X 0,Y 376.226,Z 241.621,A -85,B 0,C 180,E1 -12426.633,E2 -12426.633} C_VEL
LIN {X 0,Y 376.198,Z 241.626,A -85,B 0,C 180,E1 -12428.593,E2 -12428.593} C_VEL
LIN {X 0,Y 376.053,Z 241.644,A -85,B 0,C 180,E1 -12431.861,E2 -12431.861} C_VEL
LIN {X 0,Y 376.043,Z 241.649,A -85,B 0,C 180,E1 -12435.166,E2 -12435.166} C_VEL
LIN {X 0,Y 375.917,Z 241.665,A -85,B 0,C 180,E1 -12437.55,E2 -12437.55} C_VEL
LIN {X 0,Y 375.781,Z 241.68,A -85,B 0,C 180,E1 -12438.536,E2 -12438.536} C_VEL
LIN {X 0,Y 375.737,Z 242.188,A -85,B 0,C 180,E1 -12439.673,E2 -12439.673} C_VEL
LIN {X 0,Y 375.619,Z 245.047,A -85,B 0,C 180,E1 -12443.134,E2 -12443.134} C_VEL
LIN {X 0,Y 375.393,Z 248.095,A -85,B 0,C 180,E1 -12446.698,E2 -12446.698} C_VEL
LIN {X 0,Y 375.286,Z 250.256,A -85,B 0,C 180,E1 -12449.135,E2 -12449.135} C_VEL
LIN {X 0,Y 375.166,Z 253.667,A -85,B 0,C 180,E1 -12452.903,E2 -12452.903} C_VEL
LIN {X 0,Y 375.156,Z 254.321,A -85,B 0,C 180,E1 -12453.465,E2 -12453.465} C_VEL
LIN {X 0,Y 379.317,Z 268.149,A -85,B 0,C 180,E1 -12454.287,E2 -12454.287} C_VEL
LIN {X 0,Y 381.937,Z 279.433,A -85,B 0,C 180,E1 -12455.099,E2 -12455.099} C_VEL
LIN {X 0,Y 381.544,Z 288.043,A -85,B 0,C 180,E1 -12455.717,E2 -12455.717} C_VEL
LIN {X 0,Y 380.548,Z 299.463,A -85,B 0,C 180,E1 -12456.712,E2 -12456.712} C_VEL
LIN {X 0,Y 379.644,Z 309.513,A -85,B 0,C 180,E1 -12457.819,E2 -12457.819} C_VEL
LIN {X 0,Y 378.7,Z 319.048,A -85,B 0,C 180,E1 -12459.12,E2 -12459.12} C_VEL
LIN {X 0,Y 377.652,Z 328.111,A -85,B 0,C 180,E1 -12460.64,E2 -12460.64} C_VEL
LIN {X 0,Y 376.842,Z 335.474,A -85,B 0,C 180,E1 -12462.172,E2 -12462.172} C_VEL
LIN {X 0,Y 376.185,Z 341.493,A -85,B 0,C 180,E1 -12463.726,E2 -12463.726} C_VEL
LIN {X 0,Y 375.586,Z 346.42,A -85,B 0,C 180,E1 -12465.318,E2 -12465.318} C_VEL
LIN {X 0,Y 375.214,Z 350.269,A -85,B 0,C 180,E1 -12466.925,E2 -12466.925} C_VEL
LIN {X 0,Y 374.769,Z 353.705,A -85,B 0,C 180,E1 -12468.979,E2 -12468.979} C_VEL
LIN {X 0,Y 374.616,Z 355.188,A -85,B 0,C 180,E1 -12470.369,E2 -12470.369} C_VEL
LIN {X 0,Y 374.478,Z 356.069,A -85,B 0,C 180,E1 -12472.017,E2 -12472.017} C_VEL
LIN {X 0,Y 374.469,Z 355.96,A -85,B 0,C 180,E1 -12473.802,E2 -12473.802} C_VEL
LIN {X 0,Y 374.583,Z 354.584,A -85,B 0,C 180,E1 -12475.747,E2 -12475.747} C_VEL
LIN {X 0,Y 374.824,Z 352.157,A -85,B 0,C 180,E1 -12477.534,E2 -12477.534} C_VEL
LIN {X 0,Y 375.176,Z 347.844,A -85,B 0,C 180,E1 -12479.618,E2 -12479.618} C_VEL
LIN {X 0,Y 375.66,Z 342.161,A -85,B 0,C 180,E1 -12481.552,E2 -12481.552} C_VEL
LIN {X 0,Y 376.349,Z 335.183,A -85,B 0,C 180,E1 -12483.374,E2 -12483.374} C_VEL
LIN {X 0,Y 377.041,Z 327.754,A -85,B 0,C 180,E1 -12484.911,E2 -12484.911} C_VEL
LIN {X 0,Y 377.937,Z 318.595,A -85,B 0,C 180,E1 -12486.435,E2 -12486.435} C_VEL
LIN {X 0,Y 378.877,Z 308.164,A -85,B 0,C 180,E1 -12487.836,E2 -12487.836} C_VEL
LIN {X 0,Y 379.735,Z 297.373,A -85,B 0,C 180,E1 -12488.988,E2 -12488.988} C_VEL
LIN {X 0,Y 380.584,Z 285.052,A -85,B 0,C 180,E1 -12490.026,E2 -12490.026} C_VEL
LIN {X 0,Y 380.895,Z 277.809,A -85,B 0,C 180,E1 -12490.519,E2 -12490.519} C_VEL
LIN {X 0,Y 378.027,Z 264.545,A -85,B 0,C 180,E1 -12491.38,E2 -12491.38} C_VEL
LIN {X 0,Y 374.997,Z 252.603,A -85,B 0,C 180,E1 -12491.988,E2 -12491.988} C_VEL
LIN {X 0,Y 375.056,Z 249.819,A -85,B 0,C 180,E1 -12494.792,E2 -12494.792} C_VEL
LIN {X 0,Y 375.207,Z 246.59,A -85,B 0,C 180,E1 -12498.111,E2 -12498.111} C_VEL
LIN {X 0,Y 375.369,Z 243.439,A -85,B 0,C 180,E1 -12501.387,E2 -12501.387} C_VEL
LIN {X 0,Y 375.463,Z 242.146,A -85,B 0,C 180,E1 -12502.758,E2 -12502.758} C_VEL
LIN {X 0,Y 375.496,Z 241.715,A -85,B 0,C 180,E1 -12503.553,E2 -12503.553} C_VEL
LIN {X 0,Y 375.699,Z 241.689,A -85,B 0,C 180,E1 -12505.71,E2 -12505.71} C_VEL
LIN {X 0,Y 376.246,Z 241.618,A -85,B 0,C 180,E1 -12508.931,E2 -12508.931} C_VEL
LIN {X 0,Y 376.471,Z 241.589,A -85,B 0,C 180,E1 -12510.001,E2 -12510.001} C_VEL
LIN {X 0,Y 376.178,Z 241.629,A -85,B 0,C 180,E1 -12513.214,E2 -12513.214} C_VEL
LIN {X 0,Y 376.233,Z 241.618,A -85,B 0,C 180,E1 -12516.436,E2 -12516.436} C_VEL
LIN {X 0,Y 376.193,Z 241.624,A -85,B 0,C 180,E1 -12518.596,E2 -12518.596} C_VEL
LIN {X 0,Y 376.048,Z 241.641,A -85,B 0,C 180,E1 -12521.865,E2 -12521.865} C_VEL
LIN {X 0,Y 376.047,Z 241.646,A -85,B 0,C 180,E1 -12525.169,E2 -12525.169} C_VEL
LIN {X 0,Y 376.02,Z 241.646,A -85,B 0,C 180,E1 -12528.527,E2 -12528.527} C_VEL
LIN {X 0,Y 375.973,Z 241.65,A -85,B 0,C 180,E1 -12531.955,E2 -12531.955} C_VEL
LIN {X 0,Y 375.986,Z 241.649,A -85,B 0,C 180,E1 -12535.307,E2 -12535.307} C_VEL
LIN {X 0,Y 375.356,Z 241.731,A -85,B 0,C 180,E1 -12536.202,E2 -12536.202} C_VEL
LIN {X 0,Y 372.496,Z 242.088,A -85,B 0,C 180,E1 -12537.656,E2 -12537.656} C_VEL
LIN {X 0,Y 370.044,Z 242.393,A -85,B 0,C 180,E1 -12538.832,E2 -12538.832} C_VEL
LIN {X 0,Y 368.983,Z 242.52,A -85,B 0,C 180,E1 -12539.742,E2 -12539.742} C_VEL
LIN {X 0,Y 368.894,Z 242.531,A -85,B 0,C 180,E1 -12540.051,E2 -12540.051} C_VEL
LIN {X 0,Y 368.888,Z 242.533,A -85,B 0,C 180,E1 -12543.54,E2 -12543.54} C_VEL
LIN {X 0,Y 368.896,Z 242.536,A -85,B 0,C 180,E1 -12546.858,E2 -12546.858} C_VEL
LIN {X 0,Y 368.946,Z 242.529,A -85,B 0,C 180,E1 -12550.367,E2 -12550.367} C_VEL
LIN {X 0,Y 368.925,Z 242.528,A -85,B 0,C 180,E1 -12553.626,E2 -12553.626} C_VEL
LIN {X 0,Y 368.902,Z 242.535,A -85,B 0,C 180,E1 -12556.701,E2 -12556.701} C_VEL
LIN {X 0,Y 368.949,Z 242.525,A -85,B 0,C 180,E1 -12559.638,E2 -12559.638} C_VEL
LIN {X 0,Y 368.901,Z 242.531,A -85,B 0,C 180,E1 -12563.146,E2 -12563.146} C_VEL
LIN {X 0,Y 368.895,Z 242.537,A -85,B 0,C 180,E1 -12566.464,E2 -12566.464} C_VEL
LIN {X 0,Y 368.928,Z 242.528,A -85,B 0,C 180,E1 -12569.049,E2 -12569.049} C_VEL
LIN {X 0,Y 368.963,Z 242.524,A -85,B 0,C 180,E1 -12572.799,E2 -12572.799} C_VEL
LIN {X 0,Y 368.946,Z 242.53,A -85,B 0,C 180,E1 -12576.115,E2 -12576.115} C_VEL
LIN {X 0,Y 368.939,Z 242.531,A -85,B 0,C 180,E1 -12579.949,E2 -12579.949} C_VEL
LIN {X 0,Y 368.979,Z 242.522,A -85,B 0,C 180,E1 -12583.401,E2 -12583.401} C_VEL
LIN {X 0,Y 369.064,Z 242.511,A -85,B 0,C 180,E1 -12586.792,E2 -12586.792} C_VEL
LIN {X 0,Y 369.07,Z 242.514,A -85,B 0,C 180,E1 -12590.134,E2 -12590.134} C_VEL
LIN {X 0,Y 369.194,Z 242.497,A -85,B 0,C 180,E1 -12593.443,E2 -12593.443} C_VEL
LIN {X 0,Y 369.322,Z 242.483,A -85,B 0,C 180,E1 -12597.821,E2 -12597.821} C_VEL
LIN {X 0,Y 369.463,Z 242.464,A -85,B 0,C 180,E1 -12600.002,E2 -12600.002} C_VEL
LIN {X 0,Y 369.321,Z 242.48,A -85,B 0,C 180,E1 -12602.183,E2 -12602.183} C_VEL
LIN {X 0,Y 369.195,Z 242.494,A -85,B 0,C 180,E1 -12606.56,E2 -12606.56} C_VEL
LIN {X 0,Y 369.072,Z 242.513,A -85,B 0,C 180,E1 -12609.87,E2 -12609.87} C_VEL
LIN {X 0,Y 369.046,Z 242.516,A -85,B 0,C 180,E1 -12613.773,E2 -12613.773} C_VEL
LIN {X 0,Y 369.011,Z 242.52,A -85,B 0,C 180,E1 -12617.769,E2 -12617.769} C_VEL
LIN {X 0,Y 368.938,Z 242.531,A -85,B 0,C 180,E1 -12621.221,E2 -12621.221} C_VEL
LIN {X 0,Y 368.966,Z 242.524,A -85,B 0,C 180,E1 -12624.776,E2 -12624.776} C_VEL
LIN {X 0,Y 368.972,Z 242.527,A -85,B 0,C 180,E1 -12627.204,E2 -12627.204} C_VEL
LIN {X 0,Y 368.939,Z 242.529,A -85,B 0,C 180,E1 -12630.954,E2 -12630.954} C_VEL
LIN {X 0,Y 368.938,Z 242.531,A -85,B 0,C 180,E1 -12635.002,E2 -12635.002} C_VEL
LIN {X 0,Y 368.916,Z 242.531,A -85,B 0,C 180,E1 -12638.64,E2 -12638.64} C_VEL
LIN {X 0,Y 368.891,Z 242.535,A -85,B 0,C 180,E1 -12642.01,E2 -12642.01} C_VEL
LIN {X 0,Y 368.943,Z 242.663,A -85,B 0,C 180,E1 -12645.562,E2 -12645.562} C_VEL
LIN {X 0,Y 369.768,Z 247.028,A -85,B 0,C 180,E1 -12648.299,E2 -12648.299} C_VEL
LIN {X 0,Y 370.784,Z 253.273,A -85,B 0,C 180,E1 -12651.973,E2 -12651.973} C_VEL
LIN {X 0,Y 371.083,Z 256.988,A -85,B 0,C 180,E1 -12654.046,E2 -12654.046} C_VEL
LIN {X 0,Y 370.58,Z 261.907,A -85,B 0,C 180,E1 -12656.633,E2 -12656.633} C_VEL
LIN {X 0,Y 369.735,Z 269.296,A -85,B 0,C 180,E1 -12660.381,E2 -12660.381} C_VEL
LIN {X 0,Y 369.048,Z 276.71,A -85,B 0,C 180,E1 -12664.022,E2 -12664.022} C_VEL
LIN {X 0,Y 368.49,Z 284.09,A -85,B 0,C 180,E1 -12667.575,E2 -12667.575} C_VEL
LIN {X 0,Y 368.136,Z 290.652,A -85,B 0,C 180,E1 -12670.663,E2 -12670.663} C_VEL
LIN {X 0,Y 370.283,Z 304.039,A -85,B 0,C 180,E1 -12671.227,E2 -12671.227} C_VEL
LIN {X 0,Y 371.863,Z 316.859,A -85,B 0,C 180,E1 -12671.976,E2 -12671.976} C_VEL
LIN {X 0,Y 372.718,Z 327.052,A -85,B 0,C 180,E1 -12672.722,E2 -12672.722} C_VEL
LIN {X 0,Y 371.729,Z 339.6,A -85,B 0,C 180,E1 -12673.806,E2 -12673.806} C_VEL
LIN {X 0,Y 370.804,Z 349.519,A -85,B 0,C 180,E1 -12674.886,E2 -12674.886} C_VEL
LIN {X 0,Y 369.918,Z 359.666,A -85,B 0,C 180,E1 -12676.261,E2 -12676.261} C_VEL
LIN {X 0,Y 368.996,Z 369.429,A -85,B 0,C 180,E1 -12677.905,E2 -12677.905} C_VEL
LIN {X 0,Y 368.28,Z 377.226,A -85,B 0,C 180,E1 -12679.554,E2 -12679.554} C_VEL
LIN {X 0,Y 367.866,Z 383.478,A -85,B 0,C 180,E1 -12681.207,E2 -12681.207} C_VEL
LIN {X 0,Y 367.659,Z 388.442,A -85,B 0,C 180,E1 -12682.861,E2 -12682.861} C_VEL
LIN {X 0,Y 367.5,Z 392.254,A -85,B 0,C 180,E1 -12684.512,E2 -12684.512} C_VEL
LIN {X 0,Y 367.512,Z 394.216,A -85,B 0,C 180,E1 -12685.612,E2 -12685.612} C_VEL
LIN {X 0,Y 367.474,Z 395.749,A -85,B 0,C 180,E1 -12686.71,E2 -12686.71} C_VEL
LIN {X 0,Y 367.57,Z 396.83,A -85,B 0,C 180,E1 -12687.807,E2 -12687.807} C_VEL
LIN {X 0,Y 367.598,Z 397.495,A -85,B 0,C 180,E1 -12688.903,E2 -12688.903} C_VEL
LIN {X 0,Y 367.583,Z 397.762,A -85,B 0,C 180,E1 -12689.999,E2 -12689.999} C_VEL
LIN {X 0,Y 367.589,Z 397.636,A -85,B 0,C 180,E1 -12691.094,E2 -12691.094} C_VEL
LIN {X 0,Y 367.545,Z 397.068,A -85,B 0,C 180,E1 -12692.191,E2 -12692.191} C_VEL
LIN {X 0,Y 367.504,Z 394.712,A -85,B 0,C 180,E1 -12694.386,E2 -12694.386} C_VEL
LIN {X 0,Y 367.491,Z 391.843,A -85,B 0,C 180,E1 -12696.024,E2 -12696.024} C_VEL
LIN {X 0,Y 367.694,Z 387.897,A -85,B 0,C 180,E1 -12697.688,E2 -12697.688} C_VEL
LIN {X 0,Y 367.981,Z 382.849,A -85,B 0,C 180,E1 -12699.342,E2 -12699.342} C_VEL
LIN {X 0,Y 368.488,Z 376.532,A -85,B 0,C 180,E1 -12700.994,E2 -12700.994} C_VEL
LIN {X 0,Y 369.385,Z 368.698,A -85,B 0,C 180,E1 -12702.637,E2 -12702.637} C_VEL
LIN {X 0,Y 370.387,Z 358.921,A -85,B 0,C 180,E1 -12704.279,E2 -12704.279} C_VEL
LIN {X 0,Y 371.378,Z 348.878,A -85,B 0,C 180,E1 -12705.643,E2 -12705.643} C_VEL
LIN {X 0,Y 372.614,Z 337.593,A -85,B 0,C 180,E1 -12706.856,E2 -12706.856} C_VEL
LIN {X 0,Y 373.448,Z 328.569,A -85,B 0,C 180,E1 -12707.649,E2 -12707.649} C_VEL
LIN {X 0,Y 372.805,Z 316.923,A -85,B 0,C 180,E1 -12708.545,E2 -12708.545} C_VEL
LIN {X 0,Y 371.132,Z 304.26,A -85,B 0,C 180,E1 -12709.351,E2 -12709.351} C_VEL
LIN {X 0,Y 368.69,Z 291.526,A -85,B 0,C 180,E1 -12709.999,E2 -12709.999} C_VEL
LIN {X 0,Y 368.214,Z 289.03,A -85,B 0,C 180,E1 -12710.114,E2 -12710.114} C_VEL
LIN {X 0,Y 368.709,Z 281.308,A -85,B 0,C 180,E1 -12713.801,E2 -12713.801} C_VEL
LIN {X 0,Y 369.277,Z 274.451,A -85,B 0,C 180,E1 -12717.177,E2 -12717.177} C_VEL
LIN {X 0,Y 370.015,Z 267.306,A -85,B 0,C 180,E1 -12720.851,E2 -12720.851} C_VEL
LIN {X 0,Y 370.984,Z 260.295,A -85,B 0,C 180,E1 -12724.632,E2 -12724.632} C_VEL
LIN {X 0,Y 371.241,Z 256.858,A -85,B 0,C 180,E1 -12726.606,E2 -12726.606} C_VEL
LIN {X 0,Y 370.808,Z 253.003,A -85,B 0,C 180,E1 -12729.004,E2 -12729.004} C_VEL
LIN {X 0,Y 369.945,Z 248.344,A -85,B 0,C 180,E1 -12732.19,E2 -12732.19} C_VEL
LIN {X 0,Y 369.245,Z 244.276,A -85,B 0,C 180,E1 -12735.23,E2 -12735.23} C_VEL
LIN {X 0,Y 368.885,Z 242.539,A -85,B 0,C 180,E1 -12736.694,E2 -12736.694} C_VEL
LIN {X 0,Y 368.911,Z 242.534,A -85,B 0,C 180,E1 -12739.641,E2 -12739.641} C_VEL
LIN {X 0,Y 368.901,Z 242.536,A -85,B 0,C 180,E1 -12743.142,E2 -12743.142} C_VEL
LIN {X 0,Y 368.895,Z 242.537,A -85,B 0,C 180,E1 -12746.46,E2 -12746.46} C_VEL
LIN {X 0,Y 368.927,Z 242.533,A -85,B 0,C 180,E1 -12749.045,E2 -12749.045} C_VEL
LIN {X 0,Y 368.973,Z 242.526,A -85,B 0,C 180,E1 -12751.562,E2 -12751.562} C_VEL
LIN {X 0,Y 368.997,Z 242.523,A -85,B 0,C 180,E1 -12754.018,E2 -12754.018} C_VEL
LIN {X 0,Y 368.929,Z 242.53,A -85,B 0,C 180,E1 -12757.603,E2 -12757.603} C_VEL
LIN {X 0,Y 368.979,Z 242.525,A -85,B 0,C 180,E1 -12761.105,E2 -12761.105} C_VEL
LIN {X 0,Y 368.995,Z 242.522,A -85,B 0,C 180,E1 -12764.534,E2 -12764.534} C_VEL
LIN {X 0,Y 369.008,Z 242.521,A -85,B 0,C 180,E1 -12767.905,E2 -12767.905} C_VEL
LIN {X 0,Y 369.224,Z 242.495,A -85,B 0,C 180,E1 -12771.799,E2 -12771.799} C_VEL
LIN {X 0,Y 369.14,Z 242.504,A -85,B 0,C 180,E1 -12774.536,E2 -12774.536} C_VEL
LIN {X 0,Y 369.313,Z 242.483,A -85,B 0,C 180,E1 -12777.817,E2 -12777.817} C_VEL
LIN {X 0,Y 369.452,Z 242.466,A -85,B 0,C 180,E1 -12779.998,E2 -12779.998} C_VEL
LIN {X 0,Y 369.312,Z 242.483,A -85,B 0,C 180,E1 -12782.179,E2 -12782.179} C_VEL
LIN {X 0,Y 369.196,Z 242.497,A -85,B 0,C 180,E1 -12786.621,E2 -12786.621} C_VEL
LIN {X 0,Y 369.131,Z 242.505,A -85,B 0,C 180,E1 -12788.759,E2 -12788.759} C_VEL
LIN {X 0,Y 369.006,Z 242.522,A -85,B 0,C 180,E1 -12792.091,E2 -12792.091} C_VEL
LIN {X 0,Y 368.975,Z 242.531,A -85,B 0,C 180,E1 -12795.464,E2 -12795.464} C_VEL
LIN {X 0,Y 368.844,Z 242.546,A -85,B 0,C 180,E1 -12797.748,E2 -12797.748} C_VEL
LIN {X 0,Y 368.704,Z 242.614,A -85,B 0,C 180,E1 -12798.906,E2 -12798.906} C_VEL
LIN {X 0,Y 368.658,Z 244.48,A -85,B 0,C 180,E1 -12801.234,E2 -12801.234} C_VEL
LIN {X 0,Y 368.494,Z 247.431,A -85,B 0,C 180,E1 -12804.806,E2 -12804.806} C_VEL
LIN {X 0,Y 368.293,Z 250.579,A -85,B 0,C 180,E1 -12808.492,E2 -12808.492} C_VEL
LIN {X 0,Y 368.124,Z 253.958,A -85,B 0,C 180,E1 -12812.312,E2 -12812.312} C_VEL
LIN {X 0,Y 368.118,Z 254.583,A -85,B 0,C 180,E1 -12813.003,E2 -12813.003} C_VEL
LIN {X 0,Y 372.593,Z 269.38,A -85,B 0,C 180,E1 -12813.929,E2 -12813.929} C_VEL
LIN {X 0,Y 375.308,Z 281.21,A -85,B 0,C 180,E1 -12814.827,E2 -12814.827} C_VEL
LIN {X 0,Y 374.562,Z 292.191,A -85,B 0,C 180,E1 -12815.666,E2 -12815.666} C_VEL
LIN {X 0,Y 373.459,Z 303.818,A -85,B 0,C 180,E1 -12816.789,E2 -12816.789} C_VEL
LIN {X 0,Y 372.448,Z 314.1,A -85,B 0,C 180,E1 -12818.043,E2 -12818.043} C_VEL
LIN {X 0,Y 371.43,Z 323.208,A -85,B 0,C 180,E1 -12819.421,E2 -12819.421} C_VEL
LIN {X 0,Y 370.422,Z 331.363,A -85,B 0,C 180,E1 -12820.935,E2 -12820.935} C_VEL
LIN {X 0,Y 369.656,Z 338.024,A -85,B 0,C 180,E1 -12822.458,E2 -12822.458} C_VEL
LIN {X 0,Y 368.901,Z 344.454,A -85,B 0,C 180,E1 -12824.303,E2 -12824.303} C_VEL
LIN {X 0,Y 368.417,Z 348.661,A -85,B 0,C 180,E1 -12825.858,E2 -12825.858} C_VEL
LIN {X 0,Y 367.877,Z 352.933,A -85,B 0,C 180,E1 -12828.039,E2 -12828.039} C_VEL
LIN {X 0,Y 367.565,Z 355.239,A -85,B 0,C 180,E1 -12829.887,E2 -12829.887} C_VEL
LIN {X 0,Y 367.434,Z 356.356,A -85,B 0,C 180,E1 -12831.644,E2 -12831.644} C_VEL
LIN {X 0,Y 367.386,Z 356.416,A -85,B 0,C 180,E1 -12833.63,E2 -12833.63} C_VEL
LIN {X 0,Y 367.454,Z 355.416,A -85,B 0,C 180,E1 -12835.324,E2 -12835.324} C_VEL
LIN {X 0,Y 367.69,Z 353.127,A -85,B 0,C 180,E1 -12837.243,E2 -12837.243} C_VEL
LIN {X 0,Y 368.038,Z 349.338,A -85,B 0,C 180,E1 -12839.235,E2 -12839.235} C_VEL
LIN {X 0,Y 368.409,Z 345.22,A -85,B 0,C 180,E1 -12840.826,E2 -12840.826} C_VEL
LIN {X 0,Y 369.028,Z 338.566,A -85,B 0,C 180,E1 -12842.803,E2 -12842.803} C_VEL
LIN {X 0,Y 369.702,Z 331.797,A -85,B 0,C 180,E1 -12844.377,E2 -12844.377} C_VEL
LIN {X 0,Y 370.545,Z 323.247,A -85,B 0,C 180,E1 -12845.975,E2 -12845.975} C_VEL
LIN {X 0,Y 371.55,Z 313.264,A -85,B 0,C 180,E1 -12847.479,E2 -12847.479} C_VEL
LIN {X 0,Y 372.487,Z 303.108,A -85,B 0,C 180,E1 -12848.704,E2 -12848.704} C_VEL
LIN {X 0,Y 373.355,Z 291.991,A -85,B 0,C 180,E1 -12849.78,E2 -12849.78} C_VEL
LIN {X 0,Y 374.13,Z 279.82,A -85,B 0,C 180,E1 -12850.704,E2 -12850.704} C_VEL
LIN {X 0,Y 371.656,Z 267.679,A -85,B 0,C 180,E1 -12851.535,E2 -12851.535} C_VEL
LIN {X 0,Y 368.147,Z 254.13,A -85,B 0,C 180,E1 -12852.259,E2 -12852.259} C_VEL
LIN {X 0,Y 367.96,Z 252.959,A -85,B 0,C 180,E1 -12852.334,E2 -12852.334} C_VEL
LIN {X 0,Y 368.013,Z 249.741,A -85,B 0,C 180,E1 -12855.626,E2 -12855.626} C_VEL
LIN {X 0,Y 368.141,Z 246.503,A -85,B 0,C 180,E1 -12858.996,E2 -12858.996} C_VEL
LIN {X 0,Y 368.403,Z 242.992,A -85,B 0,C 180,E1 -12862.728,E2 -12862.728} C_VEL
LIN {X 0,Y 368.432,Z 242.595,A -85,B 0,C 180,E1 -12863.429,E2 -12863.429} C_VEL
LIN {X 0,Y 368.656,Z 242.566,A -85,B 0,C 180,E1 -12865.628,E2 -12865.628} C_VEL
LIN {X 0,Y 369.208,Z 242.495,A -85,B 0,C 180,E1 -12868.91,E2 -12868.91} C_VEL
LIN {X 0,Y 369.44,Z 242.465,A -85,B 0,C 180,E1 -12870.001,E2 -12870.001} C_VEL
LIN {X 0,Y 369.305,Z 242.48,A -85,B 0,C 180,E1 -12872.182,E2 -12872.182} C_VEL
LIN {X 0,Y 369.195,Z 242.495,A -85,B 0,C 180,E1 -12876.56,E2 -12876.56} C_VEL
LIN {X 0,Y 369.126,Z 242.505,A -85,B 0,C 180,E1 -12878.762,E2 -12878.762} C_VEL
LIN {X 0,Y 369.002,Z 242.518,A -85,B 0,C 180,E1 -12882.094,E2 -12882.094} C_VEL
LIN {X 0,Y 368.986,Z 242.523,A -85,B 0,C 180,E1 -12885.466,E2 -12885.466} C_VEL
LIN {X 0,Y 368.981,Z 242.525,A -85,B 0,C 180,E1 -12888.894,E2 -12888.894} C_VEL
LIN {X 0,Y 368.938,Z 242.527,A -85,B 0,C 180,E1 -12892.396,E2 -12892.396} C_VEL
LIN {X 0,Y 368.99,Z 242.52,A -85,B 0,C 180,E1 -12895.982,E2 -12895.982} C_VEL
LIN {X 0,Y 368.95,Z 242.53,A -85,B 0,C 180,E1 -12898.813,E2 -12898.813} C_VEL
LIN {X 0,Y 368.894,Z 242.531,A -85,B 0,C 180,E1 -12900.051,E2 -12900.051} C_VEL
LIN {X 0,Y 368.215,Z 242.621,A -85,B 0,C 180,E1 -12900.963,E2 -12900.963} C_VEL
LIN {X 0,Y 365.346,Z 242.976,A -85,B 0,C 180,E1 -12902.445,E2 -12902.445} C_VEL
LIN {X 0,Y 362.933,Z 243.275,A -85,B 0,C 180,E1 -12903.644,E2 -12903.644} C_VEL
LIN {X 0,Y 361.916,Z 243.405,A -85,B 0,C 180,E1 -12904.572,E2 -12904.572} C_VEL
LIN {X 0,Y 361.842,Z 243.409,A -85,B 0,C 180,E1 -12904.886,E2 -12904.886} C_VEL
LIN {X 0,Y 361.865,Z 243.411,A -85,B 0,C 180,E1 -12908.426,E2 -12908.426} C_VEL
LIN {X 0,Y 361.868,Z 243.407,A -85,B 0,C 180,E1 -12911.326,E2 -12911.326} C_VEL
LIN {X 0,Y 361.898,Z 243.407,A -85,B 0,C 180,E1 -12914.357,E2 -12914.357} C_VEL
LIN {X 0,Y 361.853,Z 243.409,A -85,B 0,C 180,E1 -12917.567,E2 -12917.567} C_VEL
LIN {X 0,Y 361.871,Z 243.408,A -85,B 0,C 180,E1 -12920.975,E2 -12920.975} C_VEL
LIN {X 0,Y 361.872,Z 243.41,A -85,B 0,C 180,E1 -12924.657,E2 -12924.657} C_VEL
LIN {X 0,Y 361.836,Z 243.416,A -85,B 0,C 180,E1 -12928.373,E2 -12928.373} C_VEL
LIN {X 0,Y 361.908,Z 243.407,A -85,B 0,C 180,E1 -12932.223,E2 -12932.223} C_VEL
LIN {X 0,Y 361.929,Z 243.401,A -85,B 0,C 180,E1 -12934.712,E2 -12934.712} C_VEL
LIN {X 0,Y 361.894,Z 243.408,A -85,B 0,C 180,E1 -12938.349,E2 -12938.349} C_VEL
LIN {X 0,Y 361.97,Z 243.399,A -85,B 0,C 180,E1 -12942.064,E2 -12942.064} C_VEL
LIN {X 0,Y 362.002,Z 243.395,A -85,B 0,C 180,E1 -12946.103,E2 -12946.103} C_VEL
LIN {X 0,Y 362.036,Z 243.391,A -85,B 0,C 180,E1 -12949.94,E2 -12949.94} C_VEL
LIN {X 0,Y 362.155,Z 243.372,A -85,B 0,C 180,E1 -12953.315,E2 -12953.315} C_VEL
LIN {X 0,Y 362.286,Z 243.36,A -85,B 0,C 180,E1 -12957.778,E2 -12957.778} C_VEL
LIN {X 0,Y 362.433,Z 243.34,A -85,B 0,C 180,E1 -12960.002,E2 -12960.002} C_VEL
LIN {X 0,Y 362.285,Z 243.356,A -85,B 0,C 180,E1 -12962.225,E2 -12962.225} C_VEL
LIN {X 0,Y 362.156,Z 243.371,A -85,B 0,C 180,E1 -12966.688,E2 -12966.688} C_VEL
LIN {X 0,Y 362.008,Z 243.391,A -85,B 0,C 180,E1 -12970.064,E2 -12970.064} C_VEL
LIN {X 0,Y 362.007,Z 243.392,A -85,B 0,C 180,E1 -12973.9,E2 -12973.9} C_VEL
LIN {X 0,Y 361.977,Z 243.395,A -85,B 0,C 180,E1 -12977.94,E2 -12977.94} C_VEL
LIN {X 0,Y 361.9,Z 243.406,A -85,B 0,C 180,E1 -12981.654,E2 -12981.654} C_VEL
LIN {X 0,Y 361.937,Z 243.403,A -85,B 0,C 180,E1 -12985.291,E2 -12985.291} C_VEL
LIN {X 0,Y 361.918,Z 243.402,A -85,B 0,C 180,E1 -12987.78,E2 -12987.78} C_VEL
LIN {X 0,Y 361.848,Z 243.411,A -85,B 0,C 180,E1 -12991.63,E2 -12991.63} C_VEL
LIN {X 0,Y 361.884,Z 243.409,A -85,B 0,C 180,E1 -12995.345,E2 -12995.345} C_VEL
LIN {X 0,Y 361.878,Z 243.411,A -85,B 0,C 180,E1 -12999.026,E2 -12999.026} C_VEL
LIN {X 0,Y 361.846,Z 243.414,A -85,B 0,C 180,E1 -13002.829,E2 -13002.829} C_VEL
LIN {X 0,Y 361.859,Z 243.437,A -85,B 0,C 180,E1 -13005.186,E2 -13005.186} C_VEL
LIN {X 0,Y 362.743,Z 248.044,A -85,B 0,C 180,E1 -13008.141,E2 -13008.141} C_VEL
LIN {X 0,Y 363.739,Z 254.142,A -85,B 0,C 180,E1 -13011.807,E2 -13011.807} C_VEL
LIN {X 0,Y 364.065,Z 256.638,A -85,B 0,C 180,E1 -13013.241,E2 -13013.241} C_VEL
LIN {X 0,Y 363.877,Z 260.322,A -85,B 0,C 180,E1 -13015.265,E2 -13015.265} C_VEL
LIN {X 0,Y 363.08,Z 266.472,A -85,B 0,C 180,E1 -13018.49,E2 -13018.49} C_VEL
LIN {X 0,Y 362.292,Z 273.826,A -85,B 0,C 180,E1 -13022.252,E2 -13022.252} C_VEL
LIN {X 0,Y 361.66,Z 281.327,A -85,B 0,C 180,E1 -13025.973,E2 -13025.973} C_VEL
LIN {X 0,Y 361.172,Z 288.588,A -85,B 0,C 180,E1 -13029.496,E2 -13029.496} C_VEL
LIN {X 0,Y 361.073,Z 290.277,A -85,B 0,C 180,E1 -13030.306,E2 -13030.306} C_VEL
LIN {X 0,Y 363.348,Z 304.333,A -85,B 0,C 180,E1 -13030.932,E2 -13030.932} C_VEL
LIN {X 0,Y 364.932,Z 317.399,A -85,B 0,C 180,E1 -13031.725,E2 -13031.725} C_VEL
LIN {X 0,Y 365.773,Z 327.931,A -85,B 0,C 180,E1 -13032.528,E2 -13032.528} C_VEL
LIN {X 0,Y 364.744,Z 340.225,A -85,B 0,C 180,E1 -13033.631,E2 -13033.631} C_VEL
LIN {X 0,Y 363.754,Z 350.306,A -85,B 0,C 180,E1 -13034.779,E2 -13034.779} C_VEL
LIN {X 0,Y 362.788,Z 360.828,A -85,B 0,C 180,E1 -13036.271,E2 -13036.271} C_VEL
LIN {X 0,Y 362.023,Z 368.844,A -85,B 0,C 180,E1 -13037.669,E2 -13037.669} C_VEL
LIN {X 0,Y 361.251,Z 376.691,A -85,B 0,C 180,E1 -13039.348,E2 -13039.348} C_VEL
LIN {X 0,Y 360.813,Z 382.972,A -85,B 0,C 180,E1 -13041.034,E2 -13041.034} C_VEL
LIN {X 0,Y 360.588,Z 387.961,A -85,B 0,C 180,E1 -13042.721,E2 -13042.721} C_VEL
LIN {X 0,Y 360.417,Z 391.794,A -85,B 0,C 180,E1 -13044.404,E2 -13044.404} C_VEL
LIN {X 0,Y 360.439,Z 393.767,A -85,B 0,C 180,E1 -13045.526,E2 -13045.526} C_VEL
LIN {X 0,Y 360.388,Z 395.311,A -85,B 0,C 180,E1 -13046.645,E2 -13046.645} C_VEL
LIN {X 0,Y 360.471,Z 396.408,A -85,B 0,C 180,E1 -13047.764,E2 -13047.764} C_VEL
LIN {X 0,Y 360.532,Z 397.083,A -85,B 0,C 180,E1 -13048.882,E2 -13048.882} C_VEL
LIN {X 0,Y 360.516,Z 397.358,A -85,B 0,C 180,E1 -13049.999,E2 -13049.999} C_VEL
LIN {X 0,Y 360.523,Z 397.241,A -85,B 0,C 180,E1 -13051.116,E2 -13051.116} C_VEL
LIN {X 0,Y 360.445,Z 396.688,A -85,B 0,C 180,E1 -13052.234,E2 -13052.234} C_VEL
LIN {X 0,Y 360.408,Z 394.351,A -85,B 0,C 180,E1 -13054.472,E2 -13054.472} C_VEL
LIN {X 0,Y 360.39,Z 391.84,A -85,B 0,C 180,E1 -13055.973,E2 -13055.973} C_VEL
LIN {X 0,Y 360.621,Z 387.583,A -85,B 0,C 180,E1 -13057.84,E2 -13057.84} C_VEL
LIN {X 0,Y 360.943,Z 382.559,A -85,B 0,C 180,E1 -13059.525,E2 -13059.525} C_VEL
LIN {X 0,Y 361.481,Z 376.266,A -85,B 0,C 180,E1 -13061.21,E2 -13061.21} C_VEL
LIN {X 0,Y 362.439,Z 368.478,A -85,B 0,C 180,E1 -13062.884,E2 -13062.884} C_VEL
LIN {X 0,Y 363.476,Z 358.738,A -85,B 0,C 180,E1 -13064.557,E2 -13064.557} C_VEL
LIN {X 0,Y 364.524,Z 348.743,A -85,B 0,C 180,E1 -13065.945,E2 -13065.945} C_VEL
LIN {X 0,Y 365.812,Z 337.558,A -85,B 0,C 180,E1 -13067.179,E2 -13067.179} C_VEL
LIN {X 0,Y 366.625,Z 328.683,A -85,B 0,C 180,E1 -13067.986,E2 -13067.986} C_VEL
LIN {X 0,Y 365.905,Z 316.283,A -85,B 0,C 180,E1 -13068.97,E2 -13068.97} C_VEL
LIN {X 0,Y 364.109,Z 303.19,A -85,B 0,C 180,E1 -13069.826,E2 -13069.826} C_VEL
LIN {X 0,Y 361.39,Z 289.978,A -85,B 0,C 180,E1 -13070.51,E2 -13070.51} C_VEL
LIN {X 0,Y 361.196,Z 288.611,A -85,B 0,C 180,E1 -13070.583,E2 -13070.583} C_VEL
LIN {X 0,Y 361.699,Z 281.46,A -85,B 0,C 180,E1 -13074.081,E2 -13074.081} C_VEL
LIN {X 0,Y 362.307,Z 274.231,A -85,B 0,C 180,E1 -13077.744,E2 -13077.744} C_VEL
LIN {X 0,Y 363.155,Z 266.885,A -85,B 0,C 180,E1 -13081.621,E2 -13081.621} C_VEL
LIN {X 0,Y 363.984,Z 261.286,A -85,B 0,C 180,E1 -13084.721,E2 -13084.721} C_VEL
LIN {X 0,Y 364.25,Z 257.908,A -85,B 0,C 180,E1 -13086.734,E2 -13086.734} C_VEL
LIN {X 0,Y 364.075,Z 255.61,A -85,B 0,C 180,E1 -13088.148,E2 -13088.148} C_VEL
LIN {X 0,Y 363.27,Z 251.223,A -85,B 0,C 180,E1 -13091.129,E2 -13091.129} C_VEL
LIN {X 0,Y 362.491,Z 247.003,A -85,B 0,C 180,E1 -13094.263,E2 -13094.263} C_VEL
LIN {X 0,Y 361.824,Z 243.417,A -85,B 0,C 180,E1 -13097.291,E2 -13097.291} C_VEL
LIN {X 0,Y 361.869,Z 243.412,A -85,B 0,C 180,E1 -13100.972,E2 -13100.972} C_VEL
LIN {X 0,Y 361.873,Z 243.412,A -85,B 0,C 180,E1 -13104.653,E2 -13104.653} C_VEL
LIN {X 0,Y 361.835,Z 243.415,A -85,B 0,C 180,E1 -13108.369,E2 -13108.369} C_VEL
LIN {X 0,Y 361.898,Z 243.407,A -85,B 0,C 180,E1 -13110.954,E2 -13110.954} C_VEL
LIN {X 0,Y 361.951,Z 243.401,A -85,B 0,C 180,E1 -13113.473,E2 -13113.473} C_VEL
LIN {X 0,Y 361.887,Z 243.408,A -85,B 0,C 180,E1 -13117.143,E2 -13117.143} C_VEL
LIN {X 0,Y 361.917,Z 243.404,A -85,B 0,C 180,E1 -13120.722,E2 -13120.722} C_VEL
LIN {X 0,Y 361.943,Z 243.4,A -85,B 0,C 180,E1 -13124.224,E2 -13124.224} C_VEL
LIN {X 0,Y 361.996,Z 243.395,A -85,B 0,C 180,E1 -13126.526,E2 -13126.526} C_VEL
LIN {X 0,Y 362.031,Z 243.39,A -85,B 0,C 180,E1 -13129.936,E2 -13129.936} C_VEL
LIN {X 0,Y 362.146,Z 243.376,A -85,B 0,C 180,E1 -13132.191,E2 -13132.191} C_VEL
LIN {X 0,Y 362.113,Z 243.379,A -85,B 0,C 180,E1 -13134.43,E2 -13134.43} C_VEL
LIN {X 0,Y 362.277,Z 243.36,A -85,B 0,C 180,E1 -13137.775,E2 -13137.775} C_VEL
LIN {X 0,Y 362.421,Z 243.342,A -85,B 0,C 180,E1 -13139.998,E2 -13139.998} C_VEL
LIN {X 0,Y 362.276,Z 243.36,A -85,B 0,C 180,E1 -13142.222,E2 -13142.222} C_VEL
LIN {X 0,Y 362.164,Z 243.372,A -85,B 0,C 180,E1 -13146.684,E2 -13146.684} C_VEL
LIN {X 0,Y 362.067,Z 243.385,A -85,B 0,C 180,E1 -13148.932,E2 -13148.932} C_VEL
LIN {X 0,Y 361.96,Z 243.401,A -85,B 0,C 180,E1 -13152.33,E2 -13152.33} C_VEL
LIN {X 0,Y 361.949,Z 243.405,A -85,B 0,C 180,E1 -13154.619,E2 -13154.619} C_VEL
LIN {X 0,Y 361.755,Z 243.428,A -85,B 0,C 180,E1 -13158.108,E2 -13158.108} C_VEL
LIN {X 0,Y 361.673,Z 244.875,A -85,B 0,C 180,E1 -13160.471,E2 -13160.471} C_VEL
LIN {X 0,Y 361.482,Z 247.803,A -85,B 0,C 180,E1 -13164.095,E2 -13164.095} C_VEL
LIN {X 0,Y 361.271,Z 250.941,A -85,B 0,C 180,E1 -13167.83,E2 -13167.83} C_VEL
LIN {X 0,Y 361.098,Z 254.301,A -85,B 0,C 180,E1 -13171.699,E2 -13171.699} C_VEL
LIN {X 0,Y 361.109,Z 255.225,A -85,B 0,C 180,E1 -13172.562,E2 -13172.562} C_VEL
LIN {X 0,Y 365.253,Z 268.534,A -85,B 0,C 180,E1 -13173.408,E2 -13173.408} C_VEL
LIN {X 0,Y 367.837,Z 278.772,A -85,B 0,C 180,E1 -13174.189,E2 -13174.189} C_VEL
LIN {X 0,Y 368.688,Z 283.455,A -85,B 0,C 180,E1 -13174.579,E2 -13174.579} C_VEL
LIN {X 0,Y 367.704,Z 294.561,A -85,B 0,C 180,E1 -13175.468,E2 -13175.468} C_VEL
LIN {X 0,Y 366.58,Z 305.957,A -85,B 0,C 180,E1 -13176.633,E2 -13176.633} C_VEL
LIN {X 0,Y 365.453,Z 316.321,A -85,B 0,C 180,E1 -13177.977,E2 -13177.977} C_VEL
LIN {X 0,Y 364.312,Z 326,A -85,B 0,C 180,E1 -13179.537,E2 -13179.537} C_VEL
LIN {X 0,Y 363.27,Z 333.926,A -85,B 0,C 180,E1 -13181.128,E2 -13181.128} C_VEL
LIN {X 0,Y 362.489,Z 340.356,A -85,B 0,C 180,E1 -13182.73,E2 -13182.73} C_VEL
LIN {X 0,Y 361.792,Z 345.646,A -85,B 0,C 180,E1 -13184.369,E2 -13184.369} C_VEL
LIN {X 0,Y 361.301,Z 349.84,A -85,B 0,C 180,E1 -13186.028,E2 -13186.028} C_VEL
LIN {X 0,Y 360.878,Z 353.075,A -85,B 0,C 180,E1 -13187.731,E2 -13187.731} C_VEL
LIN {X 0,Y 360.472,Z 355.809,A -85,B 0,C 180,E1 -13189.957,E2 -13189.957} C_VEL
LIN {X 0,Y 360.366,Z 356.686,A -85,B 0,C 180,E1 -13191.387,E2 -13191.387} C_VEL
LIN {X 0,Y 360.293,Z 356.908,A -85,B 0,C 180,E1 -13193.103,E2 -13193.103} C_VEL
LIN {X 0,Y 360.364,Z 356.068,A -85,B 0,C 180,E1 -13194.991,E2 -13194.991} C_VEL
LIN {X 0,Y 360.569,Z 354.006,A -85,B 0,C 180,E1 -13196.939,E2 -13196.939} C_VEL
LIN {X 0,Y 360.912,Z 350.537,A -85,B 0,C 180,E1 -13198.955,E2 -13198.955} C_VEL
LIN {X 0,Y 361.384,Z 345.272,A -85,B 0,C 180,E1 -13201.056,E2 -13201.056} C_VEL
LIN {X 0,Y 361.942,Z 339.663,A -85,B 0,C 180,E1 -13202.758,E2 -13202.758} C_VEL
LIN {X 0,Y 362.661,Z 332.64,A -85,B 0,C 180,E1 -13204.459,E2 -13204.459} C_VEL
LIN {X 0,Y 363.508,Z 324.438,A -85,B 0,C 180,E1 -13206.047,E2 -13206.047} C_VEL
LIN {X 0,Y 364.527,Z 314.794,A -85,B 0,C 180,E1 -13207.553,E2 -13207.553} C_VEL
LIN {X 0,Y 365.534,Z 304.347,A -85,B 0,C 180,E1 -13208.87,E2 -13208.87} C_VEL
LIN {X 0,Y 366.457,Z 293.044,A -85,B 0,C 180,E1 -13210,E2 -13210} C_VEL
LIN {X 0,Y 367.201,Z 281.843,A -85,B 0,C 180,E1 -13210.885,E2 -13210.885} C_VEL
LIN {X 0,Y 366.835,Z 278.47,A -85,B 0,C 180,E1 -13211.139,E2 -13211.139} C_VEL
LIN {X 0,Y 364.166,Z 266.148,A -85,B 0,C 180,E1 -13211.978,E2 -13211.978} C_VEL
LIN {X 0,Y 360.898,Z 253.334,A -85,B 0,C 180,E1 -13212.674,E2 -13212.674} C_VEL
LIN {X 0,Y 361.036,Z 249.431,A -85,B 0,C 180,E1 -13216.722,E2 -13216.722} C_VEL
LIN {X 0,Y 361.234,Z 245.35,A -85,B 0,C 180,E1 -13221.047,E2 -13221.047} C_VEL
LIN {X 0,Y 361.372,Z 243.475,A -85,B 0,C 180,E1 -13223.3,E2 -13223.3} C_VEL
LIN {X 0,Y 361.613,Z 243.444,A -85,B 0,C 180,E1 -13225.542,E2 -13225.542} C_VEL
LIN {X 0,Y 362.17,Z 243.371,A -85,B 0,C 180,E1 -13228.889,E2 -13228.889} C_VEL
LIN {X 0,Y 362.409,Z 243.34,A -85,B 0,C 180,E1 -13230.001,E2 -13230.001} C_VEL
LIN {X 0,Y 362.269,Z 243.357,A -85,B 0,C 180,E1 -13232.225,E2 -13232.225} C_VEL
LIN {X 0,Y 362.158,Z 243.372,A -85,B 0,C 180,E1 -13236.688,E2 -13236.688} C_VEL
LIN {X 0,Y 362.062,Z 243.386,A -85,B 0,C 180,E1 -13238.935,E2 -13238.935} C_VEL
LIN {X 0,Y 361.955,Z 243.396,A -85,B 0,C 180,E1 -13242.334,E2 -13242.334} C_VEL
LIN {X 0,Y 361.95,Z 243.398,A -85,B 0,C 180,E1 -13244.622,E2 -13244.622} C_VEL
LIN {X 0,Y 361.949,Z 243.397,A -85,B 0,C 180,E1 -13248.101,E2 -13248.101} C_VEL
LIN {X 0,Y 361.903,Z 243.403,A -85,B 0,C 180,E1 -13251.653,E2 -13251.653} C_VEL
LIN {X 0,Y 361.919,Z 243.403,A -85,B 0,C 180,E1 -13255.292,E2 -13255.292} C_VEL
LIN {X 0,Y 361.904,Z 243.402,A -85,B 0,C 180,E1 -13257.781,E2 -13257.781} C_VEL
LIN {X 0,Y 361.837,Z 243.412,A -85,B 0,C 180,E1 -13261.287,E2 -13261.287} C_VEL
LIN {X 0,Y 361.842,Z 243.409,A -85,B 0,C 180,E1 -13264.886,E2 -13264.886} C_VEL
LIN {X 0,Y 361.2,Z 243.491,A -85,B 0,C 180,E1 -13265.815,E2 -13265.815} C_VEL
LIN {X 0,Y 358.355,Z 243.845,A -85,B 0,C 180,E1 -13267.326,E2 -13267.326} C_VEL
LIN {X 0,Y 355.931,Z 244.151,A -85,B 0,C 180,E1 -13268.548,E2 -13268.548} C_VEL
LIN {X 0,Y 354.89,Z 244.276,A -85,B 0,C 180,E1 -13269.494,E2 -13269.494} C_VEL
LIN {X 0,Y 354.805,Z 244.285,A -85,B 0,C 180,E1 -13269.814,E2 -13269.814} C_VEL
LIN {X 0,Y 354.828,Z 244.287,A -85,B 0,C 180,E1 -13272.878,E2 -13272.878} C_VEL
LIN {X 0,Y 354.799,Z 244.289,A -85,B 0,C 180,E1 -13276.112,E2 -13276.112} C_VEL
LIN {X 0,Y 354.82,Z 244.285,A -85,B 0,C 180,E1 -13279.187,E2 -13279.187} C_VEL
LIN {X 0,Y 354.81,Z 244.291,A -85,B 0,C 180,E1 -13282.404,E2 -13282.404} C_VEL
LIN {X 0,Y 354.81,Z 244.287,A -85,B 0,C 180,E1 -13284.943,E2 -13284.943} C_VEL
LIN {X 0,Y 354.792,Z 244.293,A -85,B 0,C 180,E1 -13288.407,E2 -13288.407} C_VEL
LIN {X 0,Y 354.846,Z 244.282,A -85,B 0,C 180,E1 -13291.621,E2 -13291.621} C_VEL
LIN {X 0,Y 354.899,Z 244.28,A -85,B 0,C 180,E1 -13294.175,E2 -13294.175} C_VEL
LIN {X 0,Y 354.836,Z 244.286,A -85,B 0,C 180,E1 -13297.896,E2 -13297.896} C_VEL
LIN {X 0,Y 354.926,Z 244.275,A -85,B 0,C 180,E1 -13301.894,E2 -13301.894} C_VEL
LIN {X 0,Y 354.947,Z 244.274,A -85,B 0,C 180,E1 -13305.983,E2 -13305.983} C_VEL
LIN {X 0,Y 354.983,Z 244.268,A -85,B 0,C 180,E1 -13309.738,E2 -13309.738} C_VEL
LIN {X 0,Y 355.118,Z 244.248,A -85,B 0,C 180,E1 -13313.182,E2 -13313.182} C_VEL
LIN {X 0,Y 355.249,Z 244.236,A -85,B 0,C 180,E1 -13317.734,E2 -13317.734} C_VEL
LIN {X 0,Y 355.382,Z 244.218,A -85,B 0,C 180,E1 -13320.002,E2 -13320.002} C_VEL
LIN {X 0,Y 355.248,Z 244.232,A -85,B 0,C 180,E1 -13322.269,E2 -13322.269} C_VEL
LIN {X 0,Y 355.119,Z 244.247,A -85,B 0,C 180,E1 -13326.821,E2 -13326.821} C_VEL
LIN {X 0,Y 354.964,Z 244.267,A -85,B 0,C 180,E1 -13330.266,E2 -13330.266} C_VEL
LIN {X 0,Y 354.952,Z 244.27,A -85,B 0,C 180,E1 -13334.02,E2 -13334.02} C_VEL
LIN {X 0,Y 354.932,Z 244.271,A -85,B 0,C 180,E1 -13338.109,E2 -13338.109} C_VEL
LIN {X 0,Y 354.843,Z 244.282,A -85,B 0,C 180,E1 -13342.107,E2 -13342.107} C_VEL
LIN {X 0,Y 354.908,Z 244.275,A -85,B 0,C 180,E1 -13345.828,E2 -13345.828} C_VEL
LIN {X 0,Y 354.828,Z 244.285,A -85,B 0,C 180,E1 -13349.683,E2 -13349.683} C_VEL
LIN {X 0,Y 354.816,Z 244.286,A -85,B 0,C 180,E1 -13353.703,E2 -13353.703} C_VEL
LIN {X 0,Y 354.807,Z 244.287,A -85,B 0,C 180,E1 -13356.46,E2 -13356.46} C_VEL
LIN {X 0,Y 354.834,Z 244.287,A -85,B 0,C 180,E1 -13359.424,E2 -13359.424} C_VEL
LIN {X 0,Y 354.798,Z 244.292,A -85,B 0,C 180,E1 -13362.867,E2 -13362.867} C_VEL
LIN {X 0,Y 354.831,Z 244.432,A -85,B 0,C 180,E1 -13364.944,E2 -13364.944} C_VEL
LIN {X 0,Y 355.663,Z 248.767,A -85,B 0,C 180,E1 -13367.789,E2 -13367.789} C_VEL
LIN {X 0,Y 356.497,Z 253.766,A -85,B 0,C 180,E1 -13370.886,E2 -13370.886} C_VEL
LIN {X 0,Y 357.032,Z 257.479,A -85,B 0,C 180,E1 -13373.102,E2 -13373.102} C_VEL
LIN {X 0,Y 356.858,Z 261.167,A -85,B 0,C 180,E1 -13375.17,E2 -13375.17} C_VEL
LIN {X 0,Y 356.134,Z 266.547,A -85,B 0,C 180,E1 -13378.058,E2 -13378.058} C_VEL
LIN {X 0,Y 355.353,Z 273.424,A -85,B 0,C 180,E1 -13381.662,E2 -13381.662} C_VEL
LIN {X 0,Y 354.628,Z 281.431,A -85,B 0,C 180,E1 -13385.733,E2 -13385.733} C_VEL
LIN {X 0,Y 354.036,Z 289.66,A -85,B 0,C 180,E1 -13389.822,E2 -13389.822} C_VEL
LIN {X 0,Y 354.016,Z 289.927,A -85,B 0,C 180,E1 -13389.954,E2 -13389.954} C_VEL
LIN {X 0,Y 356.282,Z 303.933,A -85,B 0,C 180,E1 -13390.587,E2 -13390.587} C_VEL
LIN {X 0,Y 357.864,Z 316.519,A -85,B 0,C 180,E1 -13391.367,E2 -13391.367} C_VEL
LIN {X 0,Y 358.85,Z 328.753,A -85,B 0,C 180,E1 -13392.327,E2 -13392.327} C_VEL
LIN {X 0,Y 357.864,Z 339.404,A -85,B 0,C 180,E1 -13393.307,E2 -13393.307} C_VEL
LIN {X 0,Y 356.844,Z 349.579,A -85,B 0,C 180,E1 -13394.477,E2 -13394.477} C_VEL
LIN {X 0,Y 355.864,Z 360.169,A -85,B 0,C 180,E1 -13396,E2 -13396} C_VEL
LIN {X 0,Y 355.06,Z 368.22,A -85,B 0,C 180,E1 -13397.423,E2 -13397.423} C_VEL
LIN {X 0,Y 354.214,Z 376.12,A -85,B 0,C 180,E1 -13399.134,E2 -13399.134} C_VEL
LIN {X 0,Y 353.749,Z 382.435,A -85,B 0,C 180,E1 -13400.854,E2 -13400.854} C_VEL
LIN {X 0,Y 353.504,Z 387.455,A -85,B 0,C 180,E1 -13402.574,E2 -13402.574} C_VEL
LIN {X 0,Y 353.336,Z 391.317,A -85,B 0,C 180,E1 -13404.291,E2 -13404.291} C_VEL
LIN {X 0,Y 353.346,Z 393.302,A -85,B 0,C 180,E1 -13405.436,E2 -13405.436} C_VEL
LIN {X 0,Y 353.306,Z 394.859,A -85,B 0,C 180,E1 -13406.578,E2 -13406.578} C_VEL
LIN {X 0,Y 353.374,Z 395.979,A -85,B 0,C 180,E1 -13407.719,E2 -13407.719} C_VEL
LIN {X 0,Y 353.467,Z 396.667,A -85,B 0,C 180,E1 -13408.86,E2 -13408.86} C_VEL
LIN {X 0,Y 353.452,Z 396.953,A -85,B 0,C 180,E1 -13409.999,E2 -13409.999} C_VEL
LIN {X 0,Y 353.439,Z 396.845,A -85,B 0,C 180,E1 -13411.138,E2 -13411.138} C_VEL
LIN {X 0,Y 353.346,Z 396.312,A -85,B 0,C 180,E1 -13412.279,E2 -13412.279} C_VEL
LIN {X 0,Y 353.317,Z 393.995,A -85,B 0,C 180,E1 -13414.562,E2 -13414.562} C_VEL
LIN {X 0,Y 353.319,Z 391.755,A -85,B 0,C 180,E1 -13415.964,E2 -13415.964} C_VEL
LIN {X 0,Y 353.547,Z 387.269,A -85,B 0,C 180,E1 -13417.997,E2 -13417.997} C_VEL
LIN {X 0,Y 353.921,Z 382.268,A -85,B 0,C 180,E1 -13419.716,E2 -13419.716} C_VEL
LIN {X 0,Y 354.476,Z 376,A -85,B 0,C 180,E1 -13421.434,E2 -13421.434} C_VEL
